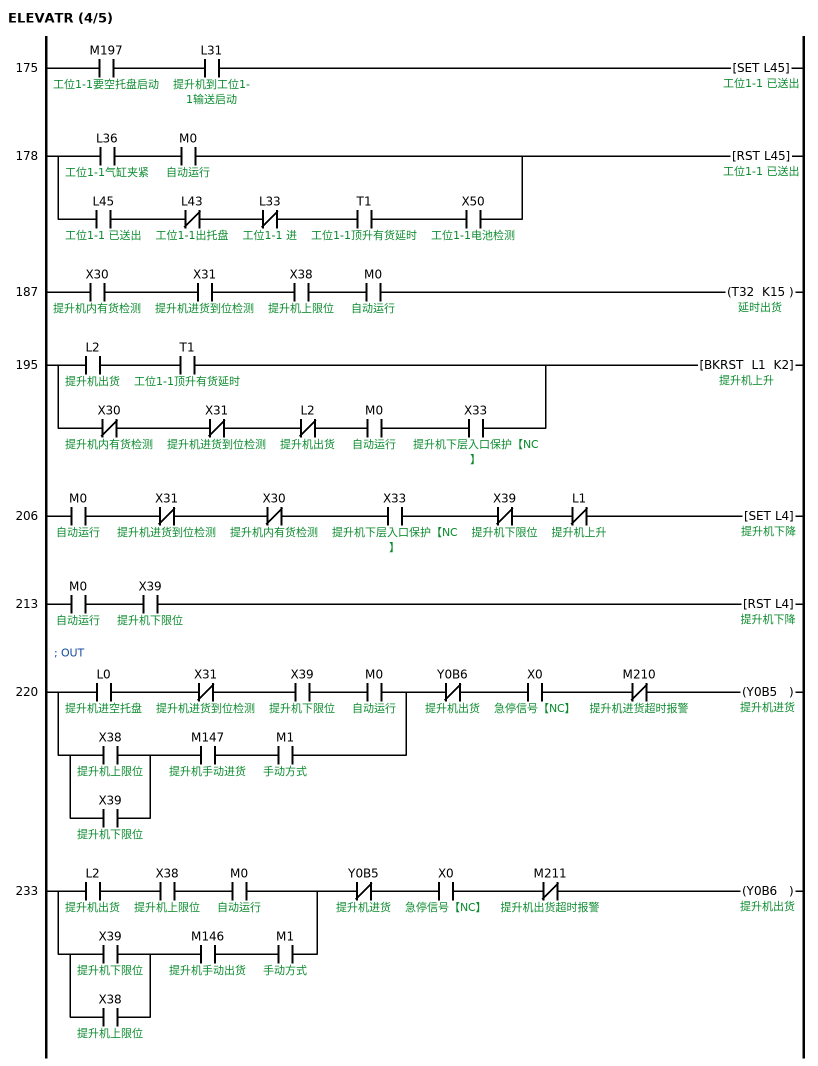
[picture p24: ladder of ELEVATR, rungs at steps 175 to 233]
175   LD      M197  ; 工位1-1要空托盘启动
      AND     L31  ; 提升机到工位1-1输送启动
      SET     L45  ; 工位1-1 已送出
178   LD      L36  ; 工位1-1气缸夹紧
      AND     M0  ; 自动运行
      LD      L45  ; 工位1-1 已送出
      ANI     L43  ; 工位1-1出托盘
      ANI     L33  ; 工位1-1 进
      AND     T1  ; 工位1-1顶升有货延时
      AND     X50  ; 工位1-1电池检测
      ORB
      RST     L45  ; 工位1-1 已送出
187   LD      X30  ; 提升机内有货检测
      AND     X31  ; 提升机进货到位检测
      AND     X38  ; 提升机上限位
      AND     M0  ; 自动运行
      OUT     T32 K15  ; 延时出货
195   LD      L2  ; 提升机出货
      AND     T1  ; 工位1-1顶升有货延时
      LDI     X30  ; 提升机内有货检测
      ANI     X31  ; 提升机进货到位检测
      ANI     L2  ; 提升机出货
      AND     M0  ; 自动运行
      AND     X33  ; 提升机下层入口保护【NC】
      ORB
      BKRST   L1 K2
206   LD      M0  ; 自动运行
      ANI     X31  ; 提升机进货到位检测
      ANI     X30  ; 提升机内有货检测
      AND     X33  ; 提升机下层入口保护【NC】
      ANI     X39  ; 提升机下限位
      ANI     L1  ; 提升机上升
      SET     L4  ; 提升机下降
213   LD      M0  ; 自动运行
      AND     X39  ; 提升机下限位
      RST     L4  ; 提升机下降
; OUT
220   LD      L0  ; 提升机进空托盘
      ANI     X31  ; 提升机进货到位检测
      AND     X39  ; 提升机下限位
      AND     M0  ; 自动运行
      LD      X38  ; 提升机上限位
      OR      X39  ; 提升机下限位
      AND     M147  ; 提升机手动进货
      AND     M1  ; 手动方式
      ORB
      ANI     Y0B6  ; 提升机出货
      AND     X0  ; 急停信号【NC】
      ANI     M210  ; 提升机进货超时报警
      OUT     Y0B5  ; 提升机进货
233   LD      L2  ; 提升机出货
      AND     X38  ; 提升机上限位
      AND     M0  ; 自动运行
      LD      X39  ; 提升机下限位
      OR      X38  ; 提升机上限位
      AND     M146  ; 提升机手动出货
      AND     M1  ; 手动方式
      ORB
      ANI     Y0B5  ; 提升机进货
      AND     X0  ; 急停信号【NC】
      ANI     M211  ; 提升机出货超时报警
      OUT     Y0B6  ; 提升机出货
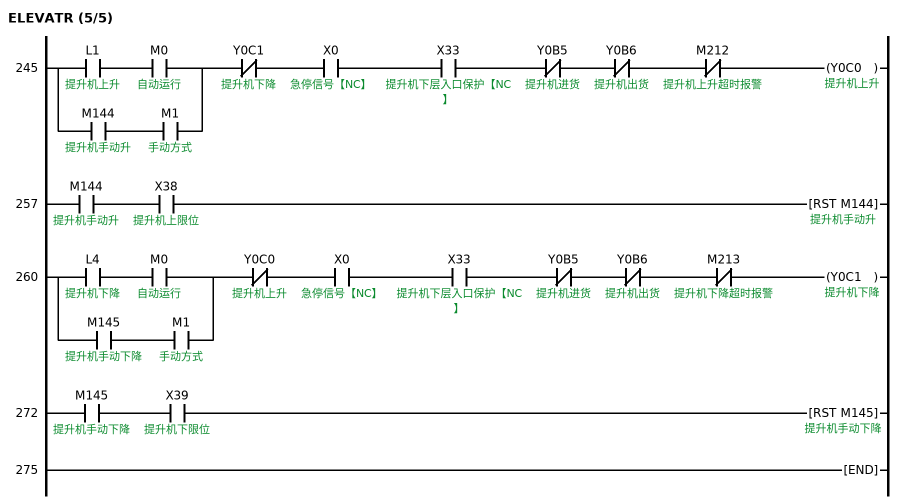
245   LD      L1  ; 提升机上升
      AND     M0  ; 自动运行
      LD      M144  ; 提升机手动升
      AND     M1  ; 手动方式
      ORB
      ANI     Y0C1  ; 提升机下降
      AND     X0  ; 急停信号【NC】
      AND     X33  ; 提升机下层入口保护【NC】
      ANI     Y0B5  ; 提升机进货
      ANI     Y0B6  ; 提升机出货
      ANI     M212  ; 提升机上升超时报警
      OUT     Y0C0  ; 提升机上升
257   LD      M144  ; 提升机手动升
      AND     X38  ; 提升机上限位
      RST     M144  ; 提升机手动升
260   LD      L4  ; 提升机下降
      AND     M0  ; 自动运行
      LD      M145  ; 提升机手动下降
      AND     M1  ; 手动方式
      ORB
      ANI     Y0C0  ; 提升机上升
      AND     X0  ; 急停信号【NC】
      AND     X33  ; 提升机下层入口保护【NC】
      ANI     Y0B5  ; 提升机进货
      ANI     Y0B6  ; 提升机出货
      ANI     M213  ; 提升机下降超时报警
      OUT     Y0C1  ; 提升机下降
272   LD      M145  ; 提升机手动下降
      AND     X39  ; 提升机下限位
      RST     M145  ; 提升机手动下降
275   END
END_PROGRAM

PROGRAM STATION1
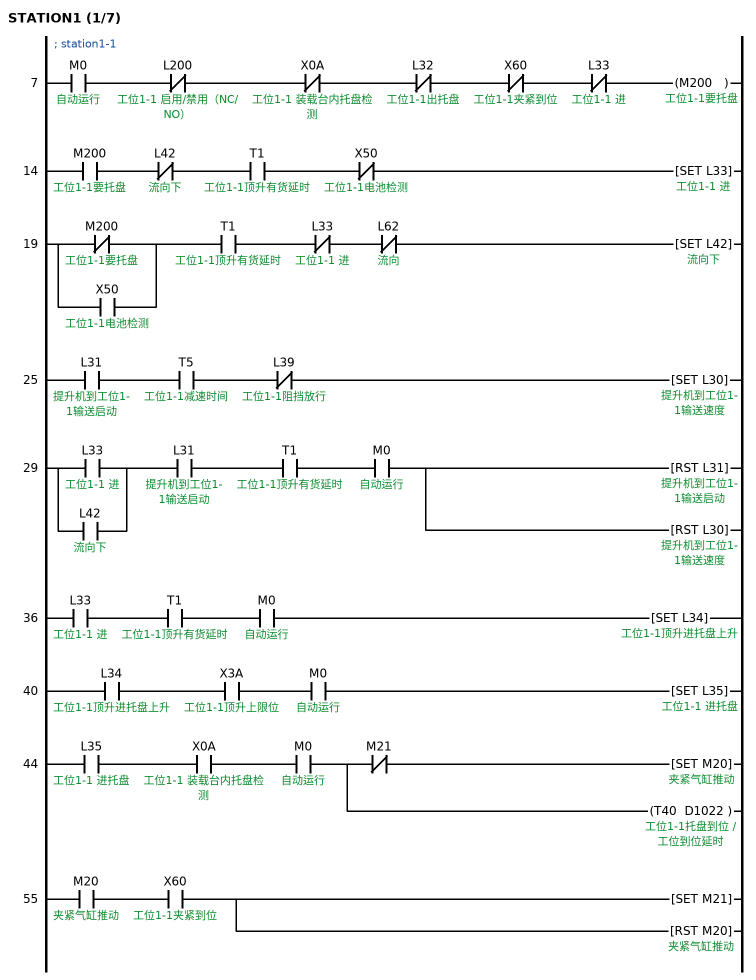
; station1-1
7     LD      M0  ; 自动运行
      ANI     L200  ; 工位1-1 启用/禁用（NC/NO）
      ANI     X0A  ; 工位1-1 装载台内托盘检测
      ANI     L32  ; 工位1-1出托盘
      ANI     X60  ; 工位1-1夹紧到位
      ANI     L33  ; 工位1-1 进
      OUT     M200  ; 工位1-1要托盘
14    LD      M200  ; 工位1-1要托盘
      ANI     L42  ; 流向下
      AND     T1  ; 工位1-1顶升有货延时
      ANI     X50  ; 工位1-1电池检测
      SET     L33  ; 工位1-1 进
19    LDI     M200  ; 工位1-1要托盘
      OR      X50  ; 工位1-1电池检测
      AND     T1  ; 工位1-1顶升有货延时
      ANI     L33  ; 工位1-1 进
      ANI     L62  ; 流向
      SET     L42  ; 流向下
25    LD      L31  ; 提升机到工位1-1输送启动
      AND     T5  ; 工位1-1减速时间
      ANI     L39  ; 工位1-1阻挡放行
      SET     L30  ; 提升机到工位1-1输送速度
29    LD      L33  ; 工位1-1 进
      OR      L42  ; 流向下
      AND     L31  ; 提升机到工位1-1输送启动
      AND     T1  ; 工位1-1顶升有货延时
      AND     M0  ; 自动运行
      RST     L31  ; 提升机到工位1-1输送启动
      RST     L30  ; 提升机到工位1-1输送速度
36    LD      L33  ; 工位1-1 进
      AND     T1  ; 工位1-1顶升有货延时
      AND     M0  ; 自动运行
      SET     L34  ; 工位1-1顶升进托盘上升
40    LD      L34  ; 工位1-1顶升进托盘上升
      AND     X3A  ; 工位1-1顶升上限位
      AND     M0  ; 自动运行
      SET     L35  ; 工位1-1 进托盘
44    LD      L35  ; 工位1-1 进托盘
      AND     X0A  ; 工位1-1 装载台内托盘检测
      AND     M0  ; 自动运行
      MPS
      ANI     M21
      SET     M20  ; 夹紧气缸推动
      MPP
      OUT     T40 D1022  ; 工位1-1托盘到位 / 工位到位延时
55    LD      M20  ; 夹紧气缸推动
      AND     X60  ; 工位1-1夹紧到位
      SET     M21
      RST     M20  ; 夹紧气缸推动
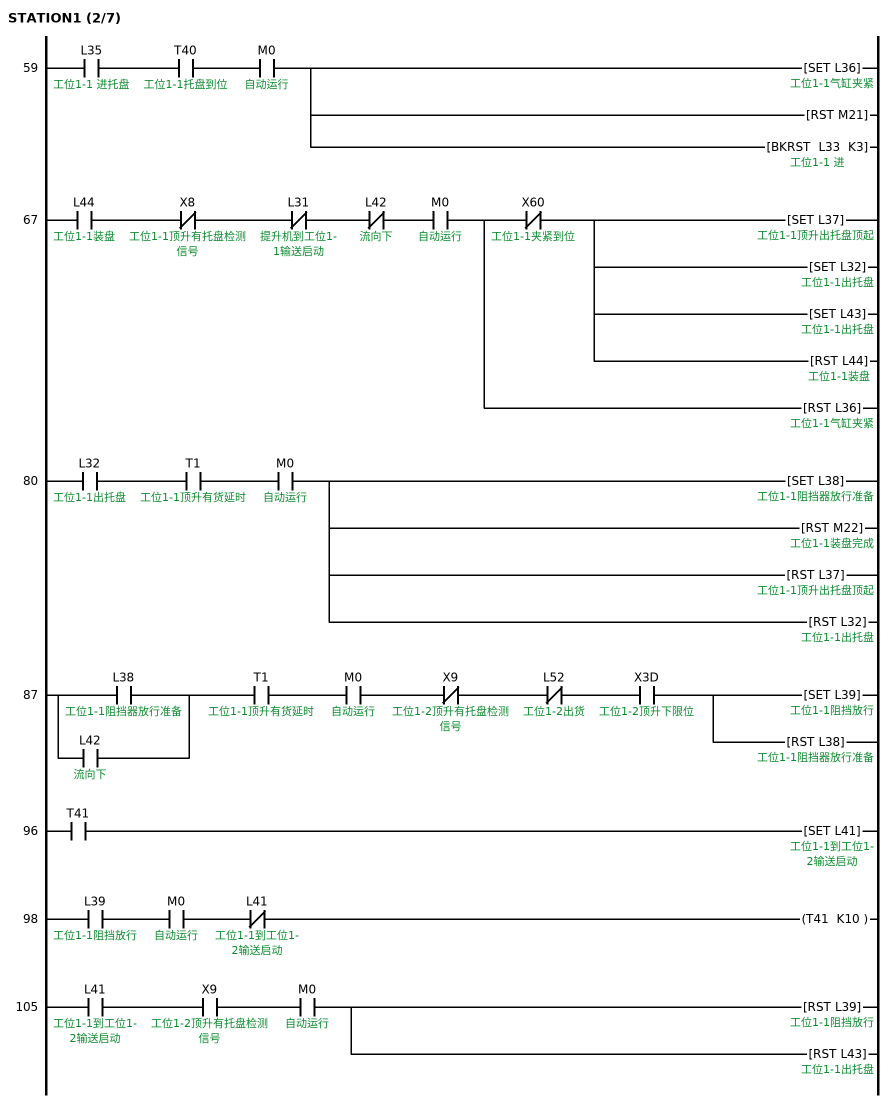
59    LD      L35  ; 工位1-1 进托盘
      AND     T40  ; 工位1-1托盘到位
      AND     M0  ; 自动运行
      SET     L36  ; 工位1-1气缸夹紧
      RST     M21
      BKRST   L33 K3
67    LD      L44  ; 工位1-1装盘
      ANI     X8  ; 工位1-1顶升有托盘检测信号
      ANI     L31  ; 提升机到工位1-1输送启动
      ANI     L42  ; 流向下
      AND     M0  ; 自动运行
      MPS
      ANI     X60  ; 工位1-1夹紧到位
      SET     L37  ; 工位1-1顶升出托盘顶起
      SET     L32  ; 工位1-1出托盘
      SET     L43  ; 工位1-1出托盘
      RST     L44  ; 工位1-1装盘
      MPP
      RST     L36  ; 工位1-1气缸夹紧
80    LD      L32  ; 工位1-1出托盘
      AND     T1  ; 工位1-1顶升有货延时
      AND     M0  ; 自动运行
      SET     L38  ; 工位1-1阻挡器放行准备
      RST     M22  ; 工位1-1装盘完成
      RST     L37  ; 工位1-1顶升出托盘顶起
      RST     L32  ; 工位1-1出托盘
87    LD      L38  ; 工位1-1阻挡器放行准备
      OR      L42  ; 流向下
      AND     T1  ; 工位1-1顶升有货延时
      AND     M0  ; 自动运行
      ANI     X9  ; 工位1-2顶升有托盘检测信号
      ANI     L52  ; 工位1-2出货
      AND     X3D  ; 工位1-2顶升下限位
      SET     L39  ; 工位1-1阻挡放行
      RST     L38  ; 工位1-1阻挡器放行准备
96    LD      T41
      SET     L41  ; 工位1-1到工位1-2输送启动
98    LD      L39  ; 工位1-1阻挡放行
      AND     M0  ; 自动运行
      ANI     L41  ; 工位1-1到工位1-2输送启动
      OUT     T41 K10
105   LD      L41  ; 工位1-1到工位1-2输送启动
      AND     X9  ; 工位1-2顶升有托盘检测信号
      AND     M0  ; 自动运行
      RST     L39  ; 工位1-1阻挡放行
      RST     L43  ; 工位1-1出托盘
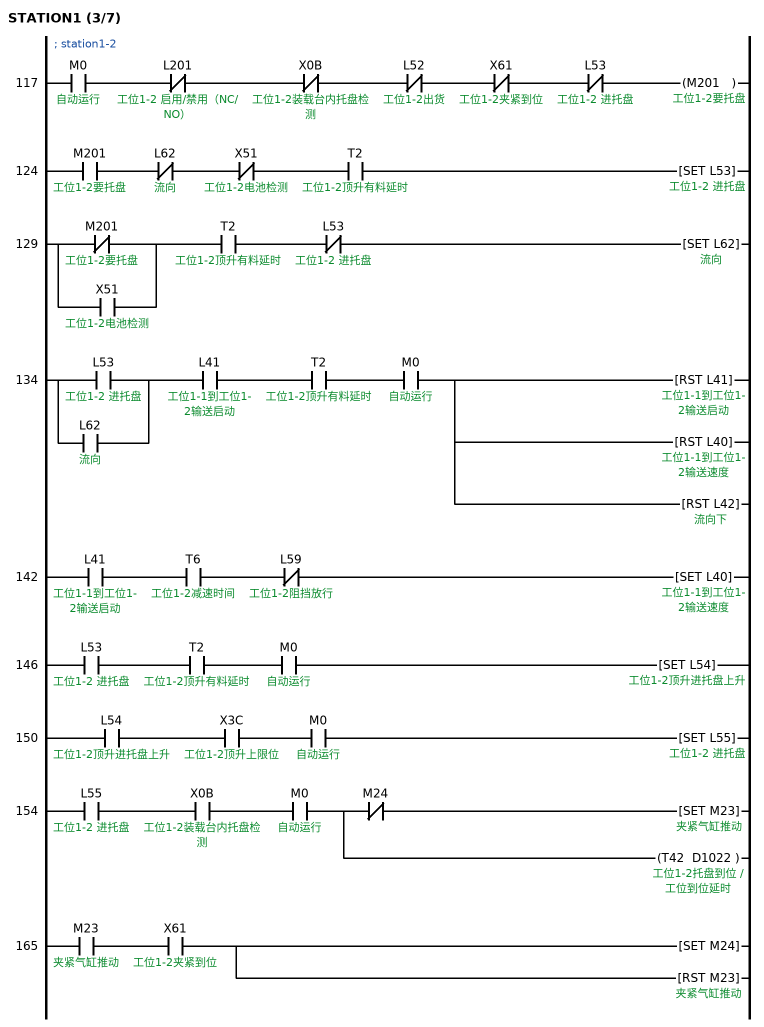
; station1-2
117   LD      M0  ; 自动运行
      ANI     L201  ; 工位1-2 启用/禁用（NC/NO）
      ANI     X0B  ; 工位1-2装载台内托盘检测
      ANI     L52  ; 工位1-2出货
      ANI     X61  ; 工位1-2夹紧到位
      ANI     L53  ; 工位1-2 进托盘
      OUT     M201  ; 工位1-2要托盘
124   LD      M201  ; 工位1-2要托盘
      ANI     L62  ; 流向
      ANI     X51  ; 工位1-2电池检测
      AND     T2  ; 工位1-2顶升有料延时
      SET     L53  ; 工位1-2 进托盘
129   LDI     M201  ; 工位1-2要托盘
      OR      X51  ; 工位1-2电池检测
      AND     T2  ; 工位1-2顶升有料延时
      ANI     L53  ; 工位1-2 进托盘
      SET     L62  ; 流向
134   LD      L53  ; 工位1-2 进托盘
      OR      L62  ; 流向
      AND     L41  ; 工位1-1到工位1-2输送启动
      AND     T2  ; 工位1-2顶升有料延时
      AND     M0  ; 自动运行
      RST     L41  ; 工位1-1到工位1-2输送启动
      RST     L40  ; 工位1-1到工位1-2输送速度
      RST     L42  ; 流向下
142   LD      L41  ; 工位1-1到工位1-2输送启动
      AND     T6  ; 工位1-2减速时间
      ANI     L59  ; 工位1-2阻挡放行
      SET     L40  ; 工位1-1到工位1-2输送速度
146   LD      L53  ; 工位1-2 进托盘
      AND     T2  ; 工位1-2顶升有料延时
      AND     M0  ; 自动运行
      SET     L54  ; 工位1-2顶升进托盘上升
150   LD      L54  ; 工位1-2顶升进托盘上升
      AND     X3C  ; 工位1-2顶升上限位
      AND     M0  ; 自动运行
      SET     L55  ; 工位1-2 进托盘
154   LD      L55  ; 工位1-2 进托盘
      AND     X0B  ; 工位1-2装载台内托盘检测
      AND     M0  ; 自动运行
      MPS
      ANI     M24
      SET     M23  ; 夹紧气缸推动
      MPP
      OUT     T42 D1022  ; 工位1-2托盘到位 / 工位到位延时
165   LD      M23  ; 夹紧气缸推动
      AND     X61  ; 工位1-2夹紧到位
      SET     M24
      RST     M23  ; 夹紧气缸推动
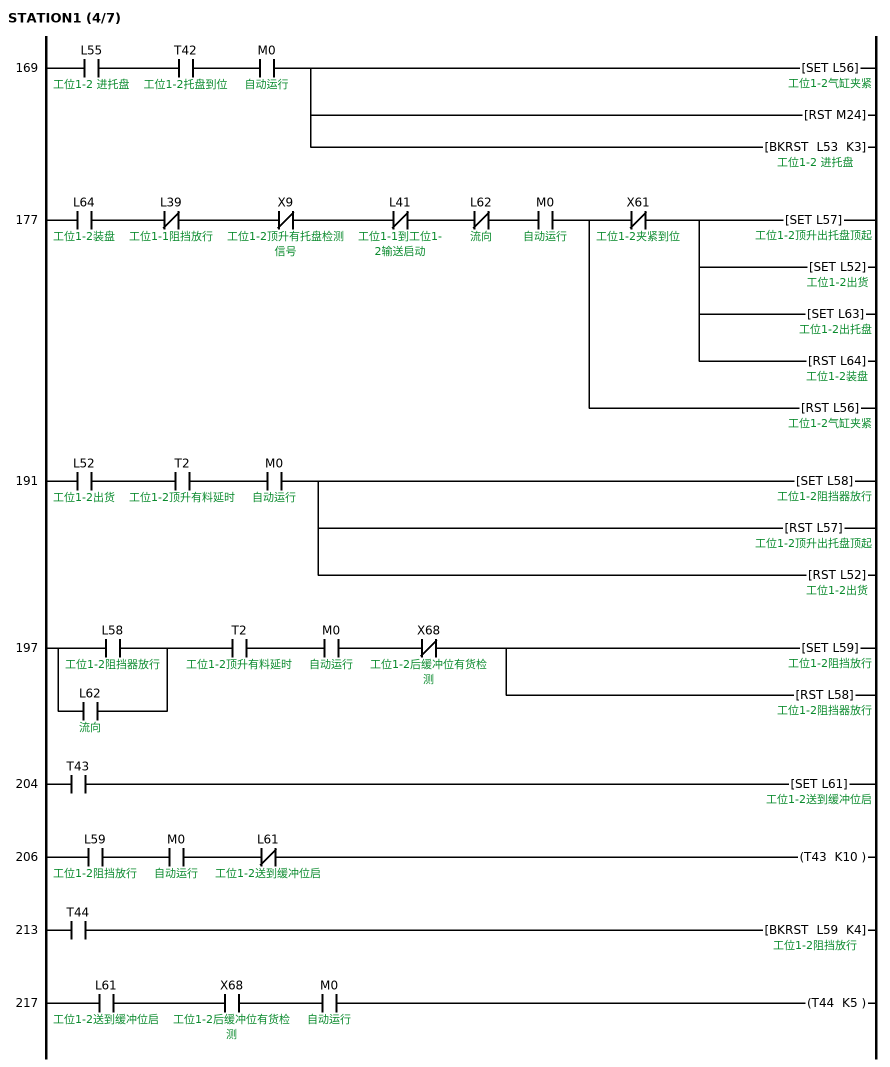
169   LD      L55  ; 工位1-2 进托盘
      AND     T42  ; 工位1-2托盘到位
      AND     M0  ; 自动运行
      SET     L56  ; 工位1-2气缸夹紧
      RST     M24
      BKRST   L53 K3
177   LD      L64  ; 工位1-2装盘
      ANI     L39  ; 工位1-1阻挡放行
      ANI     X9  ; 工位1-2顶升有托盘检测信号
      ANI     L41  ; 工位1-1到工位1-2输送启动
      ANI     L62  ; 流向
      AND     M0  ; 自动运行
      MPS
      ANI     X61  ; 工位1-2夹紧到位
      SET     L57  ; 工位1-2顶升出托盘顶起
      SET     L52  ; 工位1-2出货
      SET     L63  ; 工位1-2出托盘
      RST     L64  ; 工位1-2装盘
      MPP
      RST     L56  ; 工位1-2气缸夹紧
191   LD      L52  ; 工位1-2出货
      AND     T2  ; 工位1-2顶升有料延时
      AND     M0  ; 自动运行
      SET     L58  ; 工位1-2阻挡器放行
      RST     L57  ; 工位1-2顶升出托盘顶起
      RST     L52  ; 工位1-2出货
197   LD      L58  ; 工位1-2阻挡器放行
      OR      L62  ; 流向
      AND     T2  ; 工位1-2顶升有料延时
      AND     M0  ; 自动运行
      ANI     X68  ; 工位1-2后缓冲位有货检测
      SET     L59  ; 工位1-2阻挡放行
      RST     L58  ; 工位1-2阻挡器放行
204   LD      T43
      SET     L61  ; 工位1-2送到缓冲位启
206   LD      L59  ; 工位1-2阻挡放行
      AND     M0  ; 自动运行
      ANI     L61  ; 工位1-2送到缓冲位启
      OUT     T43 K10
213   LD      T44
      BKRST   L59 K4
217   LD      L61  ; 工位1-2送到缓冲位启
      AND     X68  ; 工位1-2后缓冲位有货检测
      AND     M0  ; 自动运行
      OUT     T44 K5
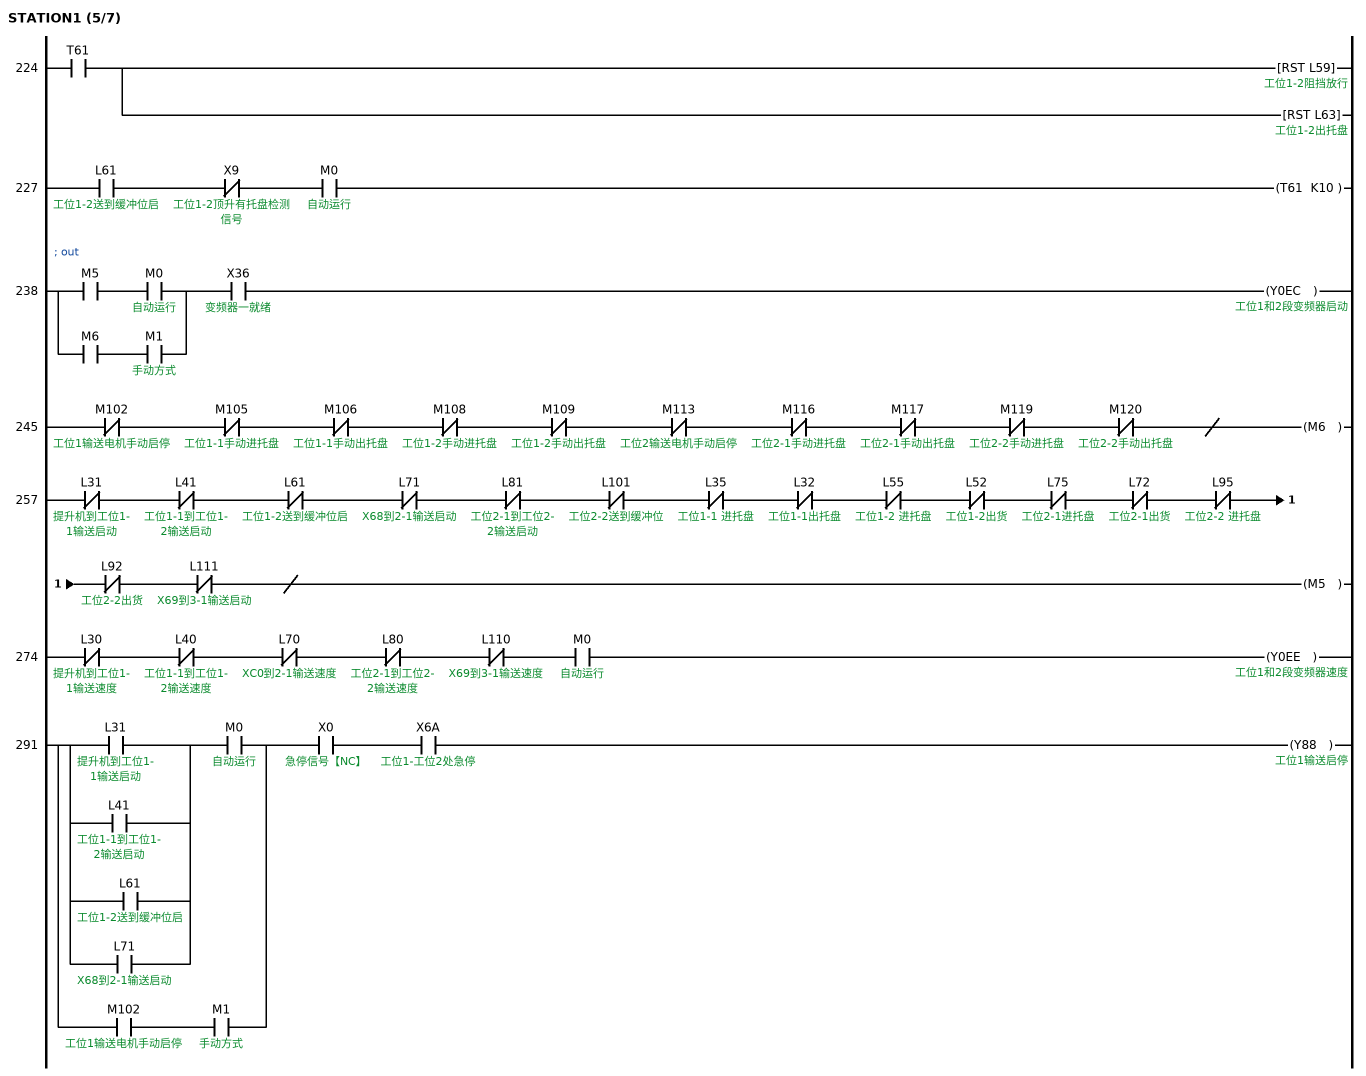
224   LD      T61
      RST     L59  ; 工位1-2阻挡放行
      RST     L63  ; 工位1-2出托盘
227   LD      L61  ; 工位1-2送到缓冲位启
      ANI     X9  ; 工位1-2顶升有托盘检测信号
      AND     M0  ; 自动运行
      OUT     T61 K10
; out
238   LD      M5
      AND     M0  ; 自动运行
      LD      M6
      AND     M1  ; 手动方式
      ORB
      AND     X36  ; 变频器一就绪
      OUT     Y0EC  ; 工位1和2段变频器启动
245   LDI     M102  ; 工位1输送电机手动启停
      ANI     M105  ; 工位1-1手动进托盘
      ANI     M106  ; 工位1-1手动出托盘
      ANI     M108  ; 工位1-2手动进托盘
      ANI     M109  ; 工位1-2手动出托盘
      ANI     M113  ; 工位2输送电机手动启停
      ANI     M116  ; 工位2-1手动进托盘
      ANI     M117  ; 工位2-1手动出托盘
      ANI     M119  ; 工位2-2手动进托盘
      ANI     M120  ; 工位2-2手动出托盘
      INV
      OUT     M6
257   LDI     L31  ; 提升机到工位1-1输送启动
      ANI     L41  ; 工位1-1到工位1-2输送启动
      ANI     L61  ; 工位1-2送到缓冲位启
      ANI     L71  ; X68到2-1输送启动
      ANI     L81  ; 工位2-1到工位2-2输送启动
      ANI     L101  ; 工位2-2送到缓冲位
      ANI     L35  ; 工位1-1 进托盘
      ANI     L32  ; 工位1-1出托盘
      ANI     L55  ; 工位1-2 进托盘
      ANI     L52  ; 工位1-2出货
      ANI     L75  ; 工位2-1进托盘
      ANI     L72  ; 工位2-1出货
      ANI     L95  ; 工位2-2 进托盘
      ANI     L92  ; 工位2-2出货
      ANI     L111  ; X69到3-1输送启动
      INV
      OUT     M5
274   LDI     L30  ; 提升机到工位1-1输送速度
      ANI     L40  ; 工位1-1到工位1-2输送速度
      ANI     L70  ; XC0到2-1输送速度
      ANI     L80  ; 工位2-1到工位2-2输送速度
      ANI     L110  ; X69到3-1输送速度
      AND     M0  ; 自动运行
      OUT     Y0EE  ; 工位1和2段变频器速度
        [note] ON高速，OFF低速
291   LD      L31  ; 提升机到工位1-1输送启动
      OR      L41  ; 工位1-1到工位1-2输送启动
      OR      L61  ; 工位1-2送到缓冲位启
      OR      L71  ; X68到2-1输送启动
      AND     M0  ; 自动运行
      LD      M102  ; 工位1输送电机手动启停
      AND     M1  ; 手动方式
      ORB
      AND     X0  ; 急停信号【NC】
      AND     X6A  ; 工位1-工位2处急停
      OUT     Y88  ; 工位1输送启停
        [note] 1-1
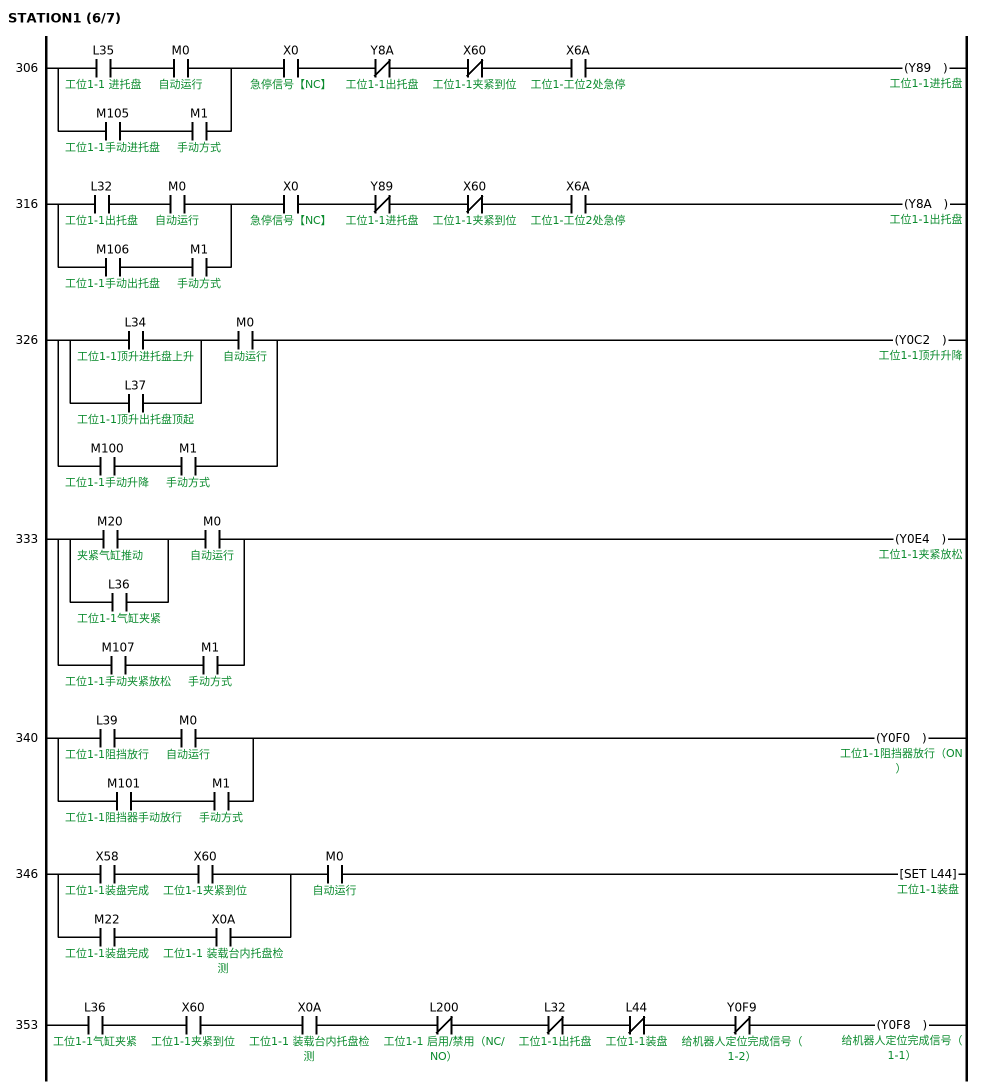
306   LD      L35  ; 工位1-1 进托盘
      AND     M0  ; 自动运行
      LD      M105  ; 工位1-1手动进托盘
      AND     M1  ; 手动方式
      ORB
      AND     X0  ; 急停信号【NC】
      ANI     Y8A  ; 工位1-1出托盘
      ANI     X60  ; 工位1-1夹紧到位
      AND     X6A  ; 工位1-工位2处急停
      OUT     Y89  ; 工位1-1进托盘
316   LD      L32  ; 工位1-1出托盘
      AND     M0  ; 自动运行
      LD      M106  ; 工位1-1手动出托盘
      AND     M1  ; 手动方式
      ORB
      AND     X0  ; 急停信号【NC】
      ANI     Y89  ; 工位1-1进托盘
      ANI     X60  ; 工位1-1夹紧到位
      AND     X6A  ; 工位1-工位2处急停
      OUT     Y8A  ; 工位1-1出托盘
326   LD      L34  ; 工位1-1顶升进托盘上升
      OR      L37  ; 工位1-1顶升出托盘顶起
      AND     M0  ; 自动运行
      LD      M100  ; 工位1-1手动升降
      AND     M1  ; 手动方式
      ORB
      OUT     Y0C2  ; 工位1-1顶升升降
333   LD      M20  ; 夹紧气缸推动
      OR      L36  ; 工位1-1气缸夹紧
      AND     M0  ; 自动运行
      LD      M107  ; 工位1-1手动夹紧放松
      AND     M1  ; 手动方式
      ORB
      OUT     Y0E4  ; 工位1-1夹紧放松
340   LD      L39  ; 工位1-1阻挡放行
      AND     M0  ; 自动运行
      LD      M101  ; 工位1-1阻挡器手动放行
      AND     M1  ; 手动方式
      ORB
      OUT     Y0F0  ; 工位1-1阻挡器放行（ON）
346   LD      X58  ; 工位1-1装盘完成
      AND     X60  ; 工位1-1夹紧到位
      LD      M22  ; 工位1-1装盘完成
      AND     X0A  ; 工位1-1 装载台内托盘检测
      ORB
      AND     M0  ; 自动运行
      SET     L44  ; 工位1-1装盘
353   LD      L36  ; 工位1-1气缸夹紧
      AND     X60  ; 工位1-1夹紧到位
      AND     X0A  ; 工位1-1 装载台内托盘检测
      ANI     L200  ; 工位1-1 启用/禁用（NC/NO）
      ANI     L32  ; 工位1-1出托盘
      ANI     L44  ; 工位1-1装盘
      ANI     Y0F9  ; 给机器人定位完成信号（1-2）
      OUT     Y0F8  ; 给机器人定位完成信号（1-1）
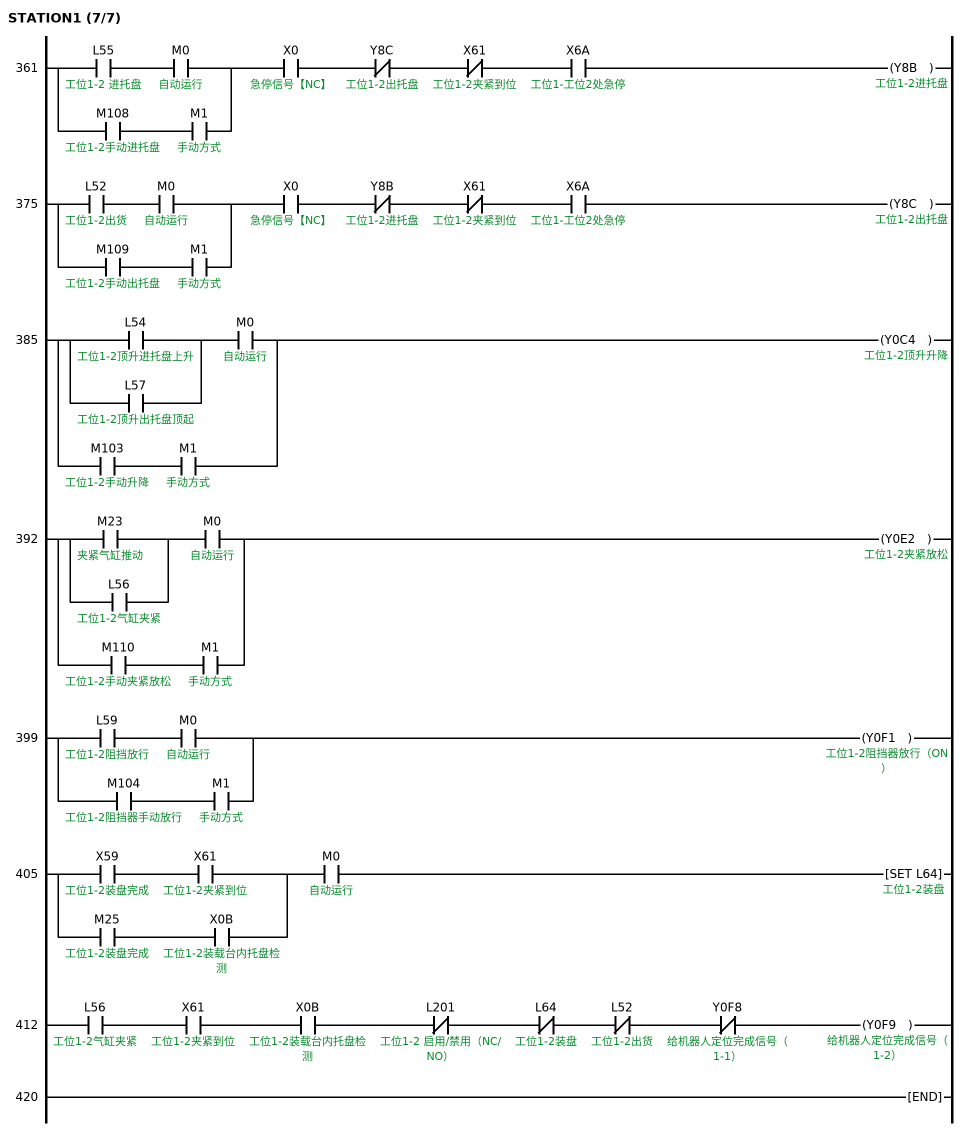
361   LD      L55  ; 工位1-2 进托盘
      AND     M0  ; 自动运行
      LD      M108  ; 工位1-2手动进托盘
      AND     M1  ; 手动方式
      ORB
      AND     X0  ; 急停信号【NC】
      ANI     Y8C  ; 工位1-2出托盘
      ANI     X61  ; 工位1-2夹紧到位
      AND     X6A  ; 工位1-工位2处急停
      OUT     Y8B  ; 工位1-2进托盘
        [note] 1-2
375   LD      L52  ; 工位1-2出货
      AND     M0  ; 自动运行
      LD      M109  ; 工位1-2手动出托盘
      AND     M1  ; 手动方式
      ORB
      AND     X0  ; 急停信号【NC】
      ANI     Y8B  ; 工位1-2进托盘
      ANI     X61  ; 工位1-2夹紧到位
      AND     X6A  ; 工位1-工位2处急停
      OUT     Y8C  ; 工位1-2出托盘
385   LD      L54  ; 工位1-2顶升进托盘上升
      OR      L57  ; 工位1-2顶升出托盘顶起
      AND     M0  ; 自动运行
      LD      M103  ; 工位1-2手动升降
      AND     M1  ; 手动方式
      ORB
      OUT     Y0C4  ; 工位1-2顶升升降
392   LD      M23  ; 夹紧气缸推动
      OR      L56  ; 工位1-2气缸夹紧
      AND     M0  ; 自动运行
      LD      M110  ; 工位1-2手动夹紧放松
      AND     M1  ; 手动方式
      ORB
      OUT     Y0E2  ; 工位1-2夹紧放松
399   LD      L59  ; 工位1-2阻挡放行
      AND     M0  ; 自动运行
      LD      M104  ; 工位1-2阻挡器手动放行
      AND     M1  ; 手动方式
      ORB
      OUT     Y0F1  ; 工位1-2阻挡器放行（ON）
405   LD      X59  ; 工位1-2装盘完成
      AND     X61  ; 工位1-2夹紧到位
      LD      M25  ; 工位1-2装盘完成
      AND     X0B  ; 工位1-2装载台内托盘检测
      ORB
      AND     M0  ; 自动运行
      SET     L64  ; 工位1-2装盘
412   LD      L56  ; 工位1-2气缸夹紧
      AND     X61  ; 工位1-2夹紧到位
      AND     X0B  ; 工位1-2装载台内托盘检测
      ANI     L201  ; 工位1-2 启用/禁用（NC/NO）
      ANI     L64  ; 工位1-2装盘
      ANI     L52  ; 工位1-2出货
      ANI     Y0F8  ; 给机器人定位完成信号（1-1）
      OUT     Y0F9  ; 给机器人定位完成信号（1-2）
420   END
END_PROGRAM

PROGRAM STATION2
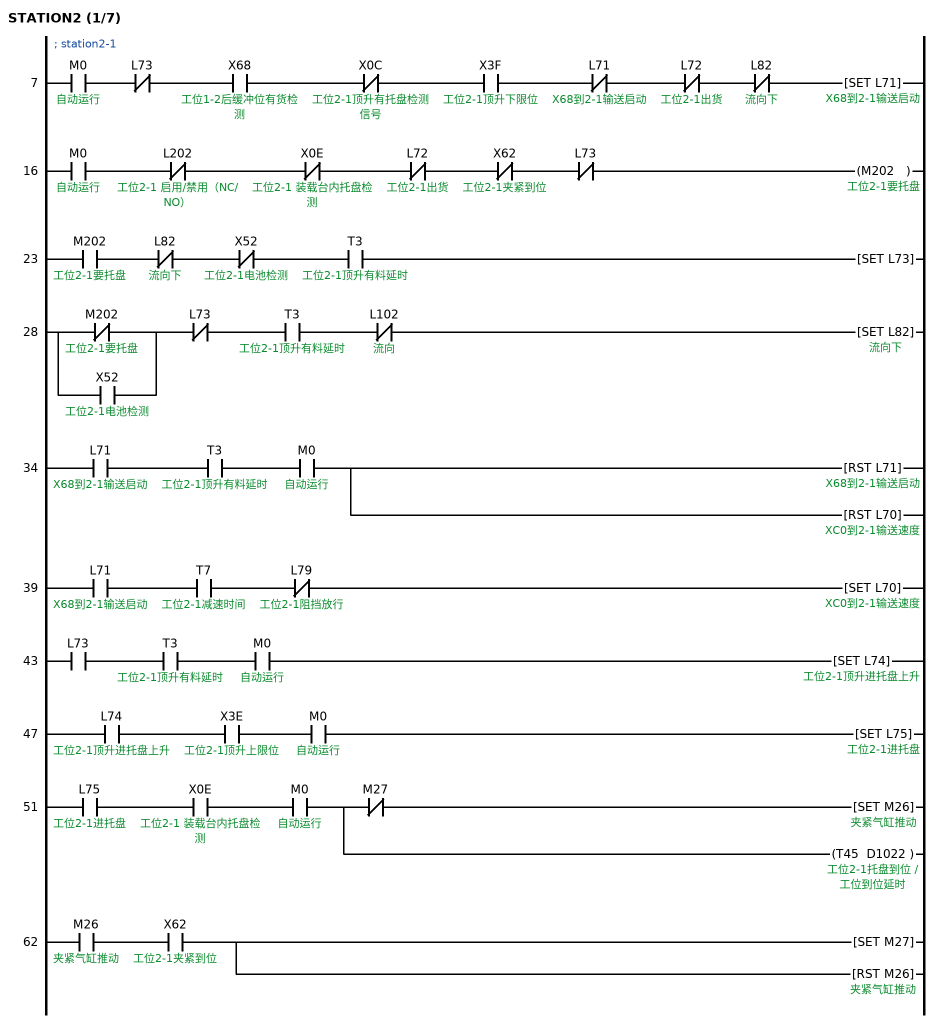
; station2-1
7     LD      M0  ; 自动运行
      ANI     L73
      AND     X68  ; 工位1-2后缓冲位有货检测
      ANI     X0C  ; 工位2-1顶升有托盘检测信号
      AND     X3F  ; 工位2-1顶升下限位
      ANI     L71  ; X68到2-1输送启动
      ANI     L72  ; 工位2-1出货
      ANI     L82  ; 流向下
      SET     L71  ; X68到2-1输送启动
16    LD      M0  ; 自动运行
      ANI     L202  ; 工位2-1 启用/禁用（NC/NO）
      ANI     X0E  ; 工位2-1 装载台内托盘检测
      ANI     L72  ; 工位2-1出货
      ANI     X62  ; 工位2-1夹紧到位
      ANI     L73
      OUT     M202  ; 工位2-1要托盘
23    LD      M202  ; 工位2-1要托盘
      ANI     L82  ; 流向下
      ANI     X52  ; 工位2-1电池检测
      AND     T3  ; 工位2-1顶升有料延时
      SET     L73
28    LDI     M202  ; 工位2-1要托盘
      OR      X52  ; 工位2-1电池检测
      ANI     L73
      AND     T3  ; 工位2-1顶升有料延时
      ANI     L102  ; 流向
      SET     L82  ; 流向下
34    LD      L71  ; X68到2-1输送启动
      AND     T3  ; 工位2-1顶升有料延时
      AND     M0  ; 自动运行
      RST     L71  ; X68到2-1输送启动
      RST     L70  ; XC0到2-1输送速度
39    LD      L71  ; X68到2-1输送启动
      AND     T7  ; 工位2-1减速时间
      ANI     L79  ; 工位2-1阻挡放行
      SET     L70  ; XC0到2-1输送速度
43    LD      L73
      AND     T3  ; 工位2-1顶升有料延时
      AND     M0  ; 自动运行
      SET     L74  ; 工位2-1顶升进托盘上升
47    LD      L74  ; 工位2-1顶升进托盘上升
      AND     X3E  ; 工位2-1顶升上限位
      AND     M0  ; 自动运行
      SET     L75  ; 工位2-1进托盘
51    LD      L75  ; 工位2-1进托盘
      AND     X0E  ; 工位2-1 装载台内托盘检测
      AND     M0  ; 自动运行
      MPS
      ANI     M27
      SET     M26  ; 夹紧气缸推动
      MPP
      OUT     T45 D1022  ; 工位2-1托盘到位 / 工位到位延时
62    LD      M26  ; 夹紧气缸推动
      AND     X62  ; 工位2-1夹紧到位
      SET     M27
      RST     M26  ; 夹紧气缸推动
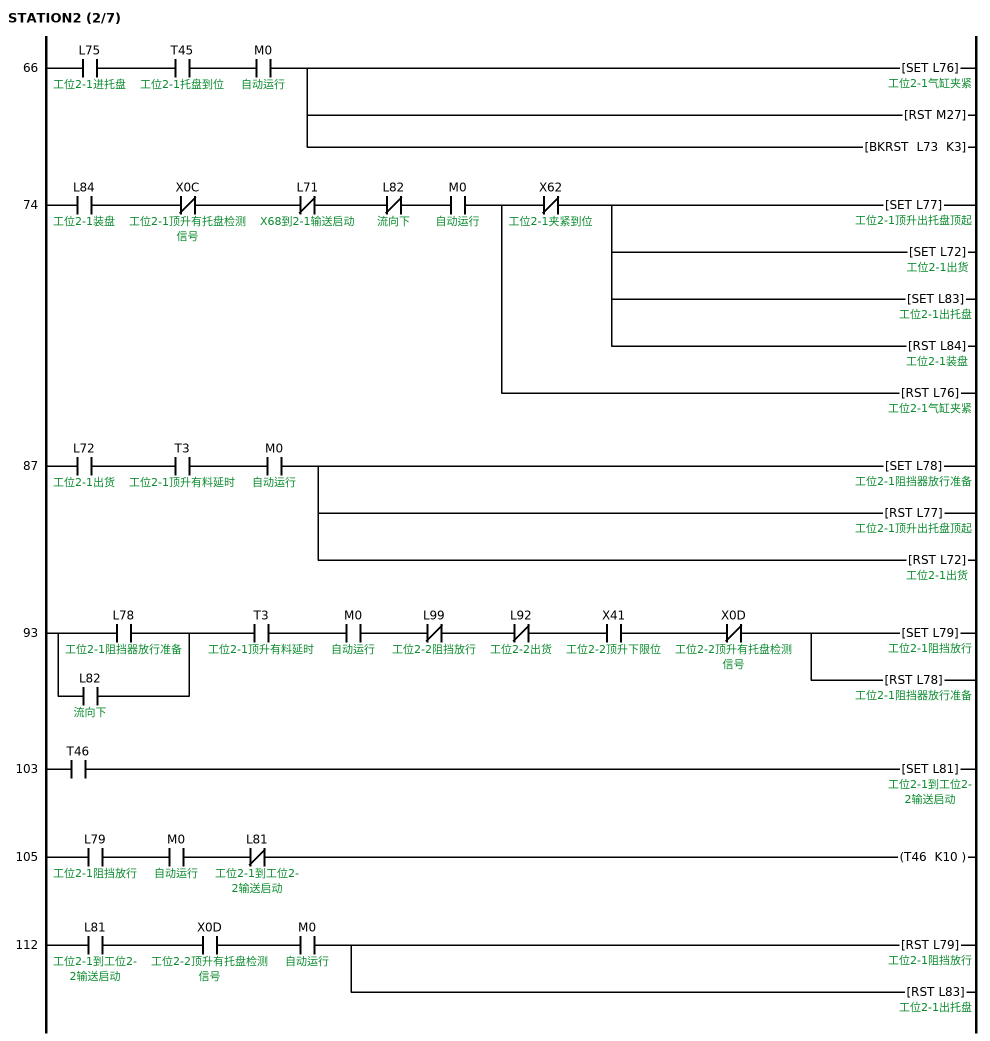
66    LD      L75  ; 工位2-1进托盘
      AND     T45  ; 工位2-1托盘到位
      AND     M0  ; 自动运行
      SET     L76  ; 工位2-1气缸夹紧
      RST     M27
      BKRST   L73 K3
74    LD      L84  ; 工位2-1装盘
      ANI     X0C  ; 工位2-1顶升有托盘检测信号
      ANI     L71  ; X68到2-1输送启动
      ANI     L82  ; 流向下
      AND     M0  ; 自动运行
      MPS
      ANI     X62  ; 工位2-1夹紧到位
      SET     L77  ; 工位2-1顶升出托盘顶起
      SET     L72  ; 工位2-1出货
      SET     L83  ; 工位2-1出托盘
      RST     L84  ; 工位2-1装盘
      MPP
      RST     L76  ; 工位2-1气缸夹紧
87    LD      L72  ; 工位2-1出货
      AND     T3  ; 工位2-1顶升有料延时
      AND     M0  ; 自动运行
      SET     L78  ; 工位2-1阻挡器放行准备
      RST     L77  ; 工位2-1顶升出托盘顶起
      RST     L72  ; 工位2-1出货
93    LD      L78  ; 工位2-1阻挡器放行准备
      OR      L82  ; 流向下
      AND     T3  ; 工位2-1顶升有料延时
      AND     M0  ; 自动运行
      ANI     L99  ; 工位2-2阻挡放行
      ANI     L92  ; 工位2-2出货
      AND     X41  ; 工位2-2顶升下限位
      ANI     X0D  ; 工位2-2顶升有托盘检测信号
      SET     L79  ; 工位2-1阻挡放行
      RST     L78  ; 工位2-1阻挡器放行准备
103   LD      T46
      SET     L81  ; 工位2-1到工位2-2输送启动
105   LD      L79  ; 工位2-1阻挡放行
      AND     M0  ; 自动运行
      ANI     L81  ; 工位2-1到工位2-2输送启动
      OUT     T46 K10
112   LD      L81  ; 工位2-1到工位2-2输送启动
      AND     X0D  ; 工位2-2顶升有托盘检测信号
      AND     M0  ; 自动运行
      RST     L79  ; 工位2-1阻挡放行
      RST     L83  ; 工位2-1出托盘
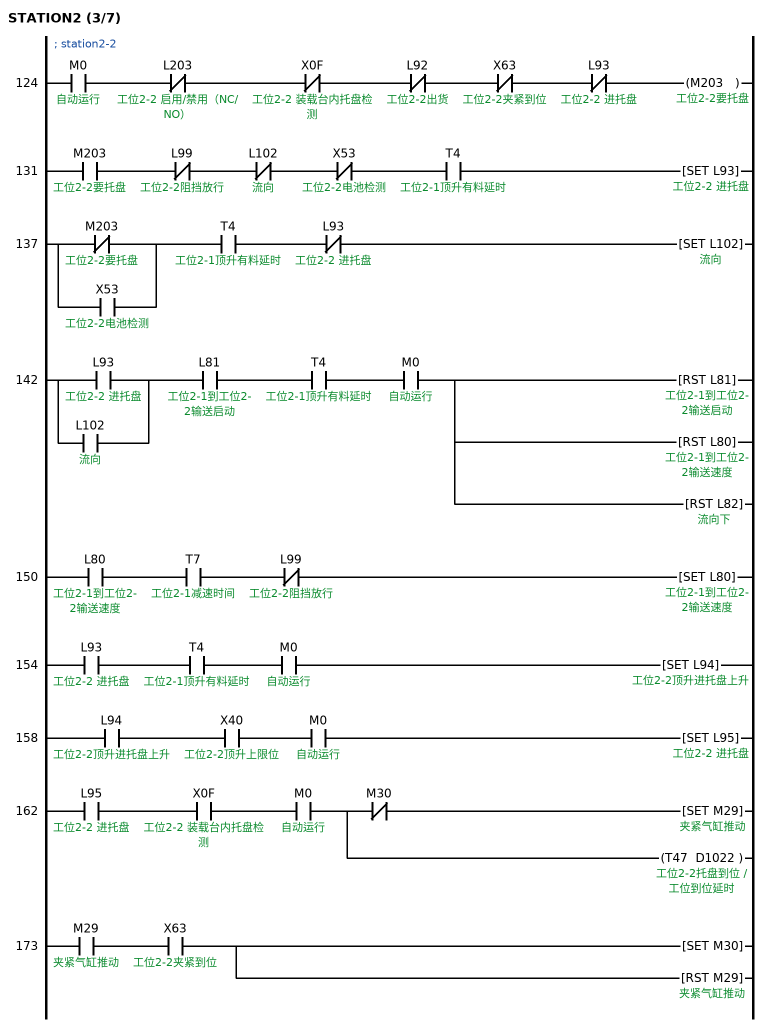
; station2-2
124   LD      M0  ; 自动运行
      ANI     L203  ; 工位2-2 启用/禁用（NC/NO）
      ANI     X0F  ; 工位2-2 装载台内托盘检测
      ANI     L92  ; 工位2-2出货
      ANI     X63  ; 工位2-2夹紧到位
      ANI     L93  ; 工位2-2 进托盘
      OUT     M203  ; 工位2-2要托盘
131   LD      M203  ; 工位2-2要托盘
      ANI     L99  ; 工位2-2阻挡放行
      ANI     L102  ; 流向
      ANI     X53  ; 工位2-2电池检测
      AND     T4  ; 工位2-1顶升有料延时
      SET     L93  ; 工位2-2 进托盘
137   LDI     M203  ; 工位2-2要托盘
      OR      X53  ; 工位2-2电池检测
      AND     T4  ; 工位2-1顶升有料延时
      ANI     L93  ; 工位2-2 进托盘
      SET     L102  ; 流向
142   LD      L93  ; 工位2-2 进托盘
      OR      L102  ; 流向
      AND     L81  ; 工位2-1到工位2-2输送启动
      AND     T4  ; 工位2-1顶升有料延时
      AND     M0  ; 自动运行
      RST     L81  ; 工位2-1到工位2-2输送启动
      RST     L80  ; 工位2-1到工位2-2输送速度
      RST     L82  ; 流向下
150   LD      L80  ; 工位2-1到工位2-2输送速度
      AND     T7  ; 工位2-1减速时间
      ANI     L99  ; 工位2-2阻挡放行
      SET     L80  ; 工位2-1到工位2-2输送速度
154   LD      L93  ; 工位2-2 进托盘
      AND     T4  ; 工位2-1顶升有料延时
      AND     M0  ; 自动运行
      SET     L94  ; 工位2-2顶升进托盘上升
158   LD      L94  ; 工位2-2顶升进托盘上升
      AND     X40  ; 工位2-2顶升上限位
      AND     M0  ; 自动运行
      SET     L95  ; 工位2-2 进托盘
162   LD      L95  ; 工位2-2 进托盘
      AND     X0F  ; 工位2-2 装载台内托盘检测
      AND     M0  ; 自动运行
      MPS
      ANI     M30
      SET     M29  ; 夹紧气缸推动
      MPP
      OUT     T47 D1022  ; 工位2-2托盘到位 / 工位到位延时
173   LD      M29  ; 夹紧气缸推动
      AND     X63  ; 工位2-2夹紧到位
      SET     M30
      RST     M29  ; 夹紧气缸推动
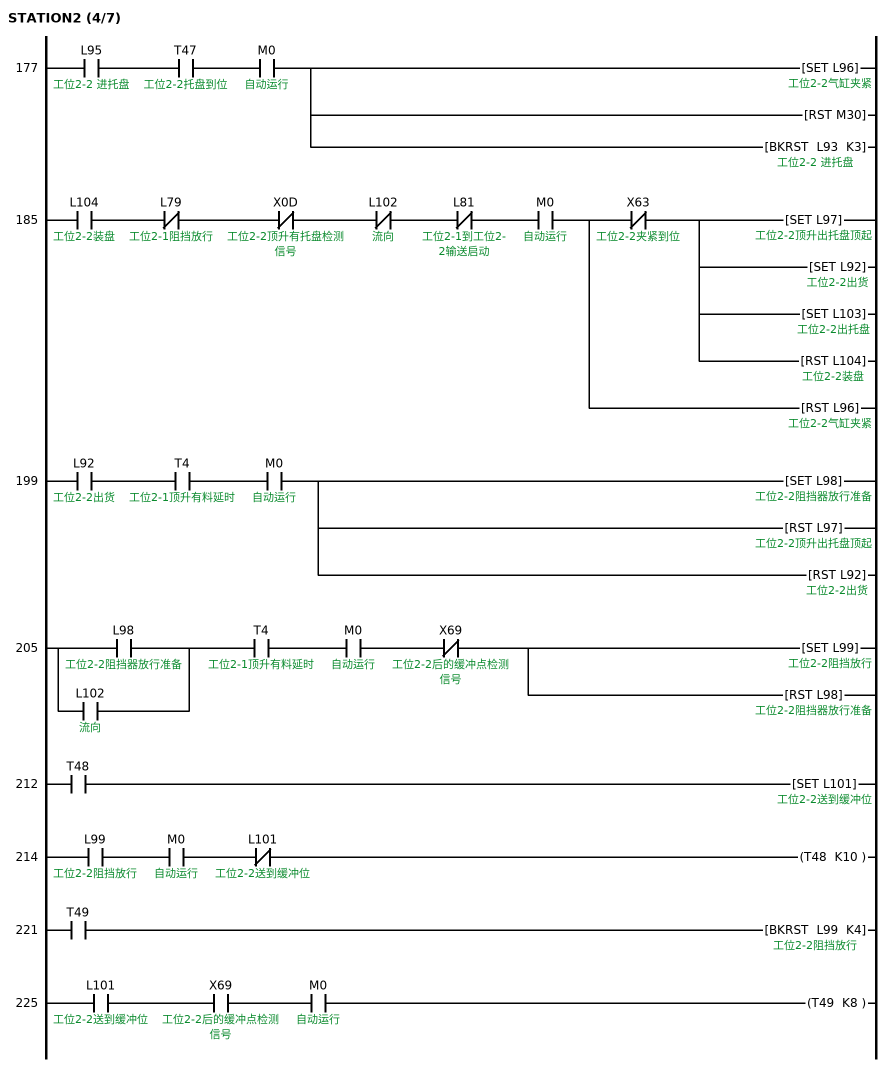
177   LD      L95  ; 工位2-2 进托盘
      AND     T47  ; 工位2-2托盘到位
      AND     M0  ; 自动运行
      SET     L96  ; 工位2-2气缸夹紧
      RST     M30
      BKRST   L93 K3
185   LD      L104  ; 工位2-2装盘
      ANI     L79  ; 工位2-1阻挡放行
      ANI     X0D  ; 工位2-2顶升有托盘检测信号
      ANI     L102  ; 流向
      ANI     L81  ; 工位2-1到工位2-2输送启动
      AND     M0  ; 自动运行
      MPS
      ANI     X63  ; 工位2-2夹紧到位
      SET     L97  ; 工位2-2顶升出托盘顶起
      SET     L92  ; 工位2-2出货
      SET     L103  ; 工位2-2出托盘
      RST     L104  ; 工位2-2装盘
      MPP
      RST     L96  ; 工位2-2气缸夹紧
199   LD      L92  ; 工位2-2出货
      AND     T4  ; 工位2-1顶升有料延时
      AND     M0  ; 自动运行
      SET     L98  ; 工位2-2阻挡器放行准备
      RST     L97  ; 工位2-2顶升出托盘顶起
      RST     L92  ; 工位2-2出货
205   LD      L98  ; 工位2-2阻挡器放行准备
      OR      L102  ; 流向
      AND     T4  ; 工位2-1顶升有料延时
      AND     M0  ; 自动运行
      ANI     X69  ; 工位2-2后的缓冲点检测信号
      SET     L99  ; 工位2-2阻挡放行
      RST     L98  ; 工位2-2阻挡器放行准备
212   LD      T48
      SET     L101  ; 工位2-2送到缓冲位
214   LD      L99  ; 工位2-2阻挡放行
      AND     M0  ; 自动运行
      ANI     L101  ; 工位2-2送到缓冲位
      OUT     T48 K10
221   LD      T49
      BKRST   L99 K4
225   LD      L101  ; 工位2-2送到缓冲位
      AND     X69  ; 工位2-2后的缓冲点检测信号
      AND     M0  ; 自动运行
      OUT     T49 K8
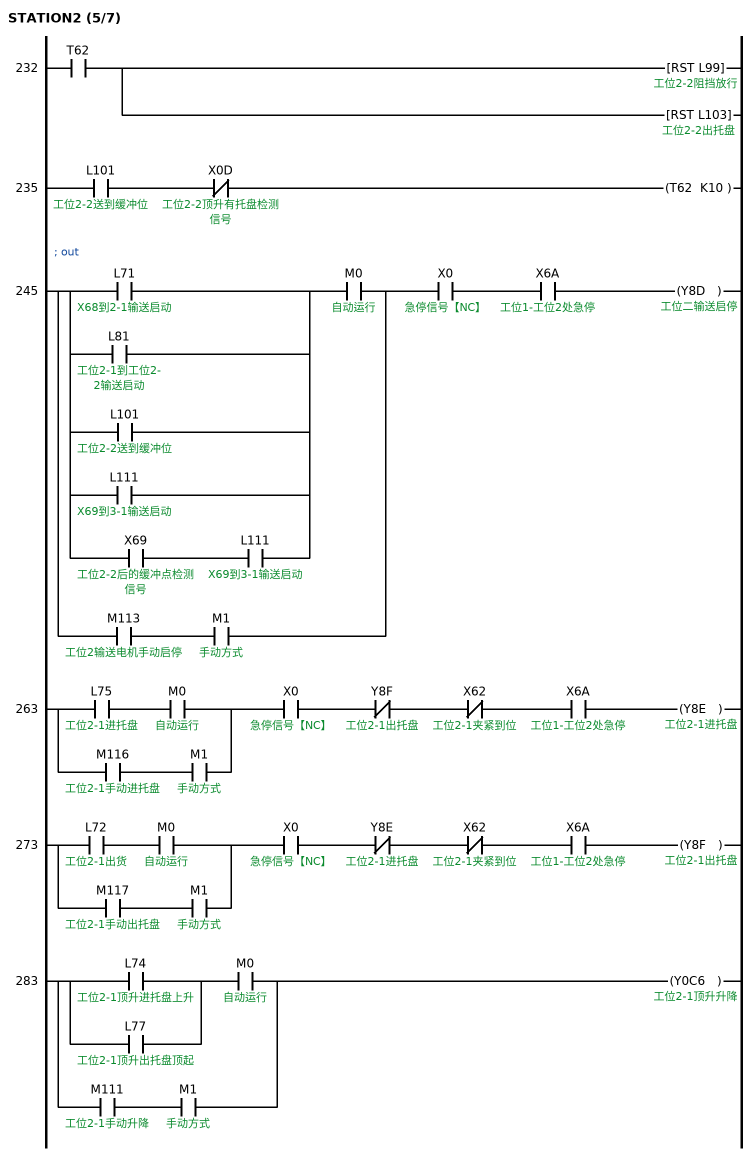
232   LD      T62
      RST     L99  ; 工位2-2阻挡放行
      RST     L103  ; 工位2-2出托盘
235   LD      L101  ; 工位2-2送到缓冲位
      ANI     X0D  ; 工位2-2顶升有托盘检测信号
      OUT     T62 K10
; out
245   LD      L71  ; X68到2-1输送启动
      OR      L81  ; 工位2-1到工位2-2输送启动
      OR      L101  ; 工位2-2送到缓冲位
      OR      L111  ; X69到3-1输送启动
      LD      X69  ; 工位2-2后的缓冲点检测信号
      AND     L111  ; X69到3-1输送启动
      ORB
      AND     M0  ; 自动运行
      LD      M113  ; 工位2输送电机手动启停
      AND     M1  ; 手动方式
      ORB
      AND     X0  ; 急停信号【NC】
      AND     X6A  ; 工位1-工位2处急停
      OUT     Y8D  ; 工位二输送启停
        [note] 1-1
263   LD      L75  ; 工位2-1进托盘
      AND     M0  ; 自动运行
      LD      M116  ; 工位2-1手动进托盘
      AND     M1  ; 手动方式
      ORB
      AND     X0  ; 急停信号【NC】
      ANI     Y8F  ; 工位2-1出托盘
      ANI     X62  ; 工位2-1夹紧到位
      AND     X6A  ; 工位1-工位2处急停
      OUT     Y8E  ; 工位2-1进托盘
273   LD      L72  ; 工位2-1出货
      AND     M0  ; 自动运行
      LD      M117  ; 工位2-1手动出托盘
      AND     M1  ; 手动方式
      ORB
      AND     X0  ; 急停信号【NC】
      ANI     Y8E  ; 工位2-1进托盘
      ANI     X62  ; 工位2-1夹紧到位
      AND     X6A  ; 工位1-工位2处急停
      OUT     Y8F  ; 工位2-1出托盘
283   LD      L74  ; 工位2-1顶升进托盘上升
      OR      L77  ; 工位2-1顶升出托盘顶起
      AND     M0  ; 自动运行
      LD      M111  ; 工位2-1手动升降
      AND     M1  ; 手动方式
      ORB
      OUT     Y0C6  ; 工位2-1顶升升降
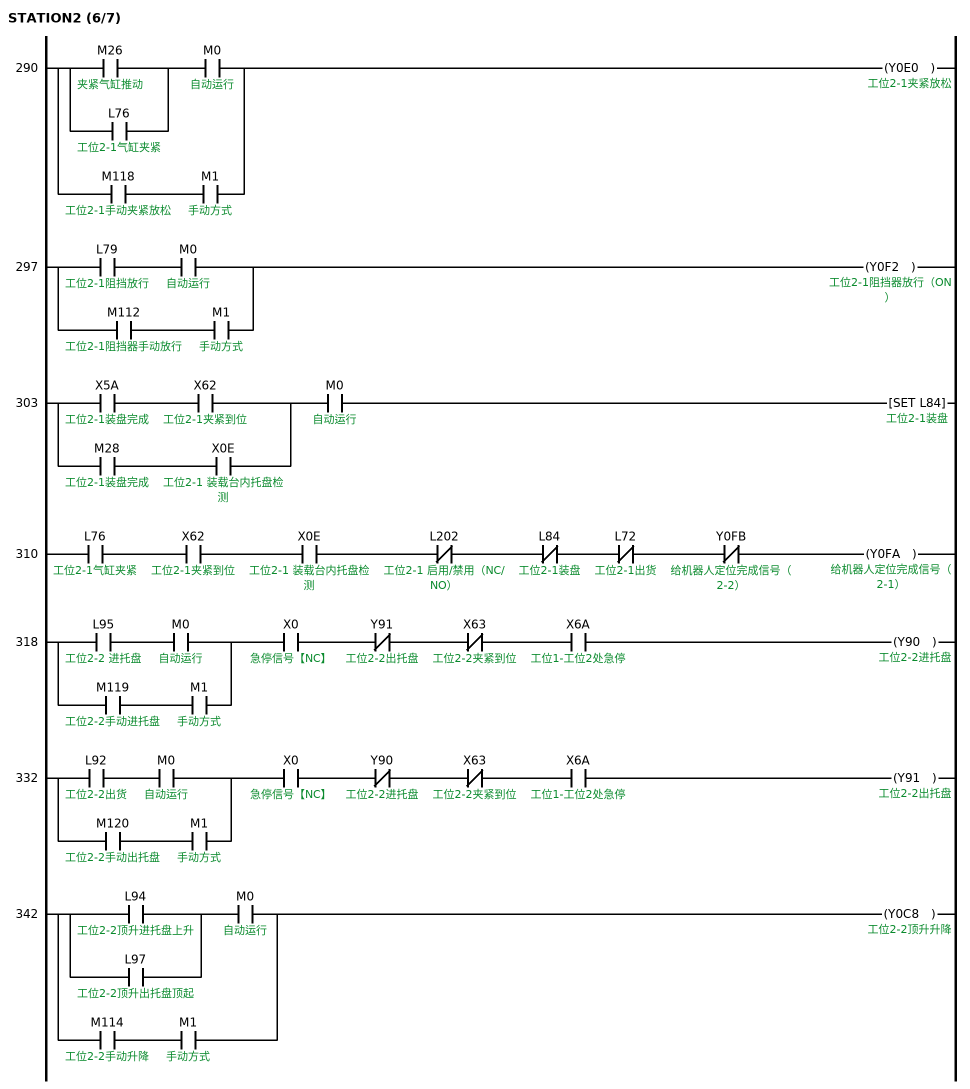
290   LD      M26  ; 夹紧气缸推动
      OR      L76  ; 工位2-1气缸夹紧
      AND     M0  ; 自动运行
      LD      M118  ; 工位2-1手动夹紧放松
      AND     M1  ; 手动方式
      ORB
      OUT     Y0E0  ; 工位2-1夹紧放松
297   LD      L79  ; 工位2-1阻挡放行
      AND     M0  ; 自动运行
      LD      M112  ; 工位2-1阻挡器手动放行
      AND     M1  ; 手动方式
      ORB
      OUT     Y0F2  ; 工位2-1阻挡器放行（ON）
303   LD      X5A  ; 工位2-1装盘完成
      AND     X62  ; 工位2-1夹紧到位
      LD      M28  ; 工位2-1装盘完成
      AND     X0E  ; 工位2-1 装载台内托盘检测
      ORB
      AND     M0  ; 自动运行
      SET     L84  ; 工位2-1装盘
310   LD      L76  ; 工位2-1气缸夹紧
      AND     X62  ; 工位2-1夹紧到位
      AND     X0E  ; 工位2-1 装载台内托盘检测
      ANI     L202  ; 工位2-1 启用/禁用（NC/NO）
      ANI     L84  ; 工位2-1装盘
      ANI     L72  ; 工位2-1出货
      ANI     Y0FB  ; 给机器人定位完成信号（2-2）
      OUT     Y0FA  ; 给机器人定位完成信号（2-1）
318   LD      L95  ; 工位2-2 进托盘
      AND     M0  ; 自动运行
      LD      M119  ; 工位2-2手动进托盘
      AND     M1  ; 手动方式
      ORB
      AND     X0  ; 急停信号【NC】
      ANI     Y91  ; 工位2-2出托盘
      ANI     X63  ; 工位2-2夹紧到位
      AND     X6A  ; 工位1-工位2处急停
      OUT     Y90  ; 工位2-2进托盘
        [note] 1-2
332   LD      L92  ; 工位2-2出货
      AND     M0  ; 自动运行
      LD      M120  ; 工位2-2手动出托盘
      AND     M1  ; 手动方式
      ORB
      AND     X0  ; 急停信号【NC】
      ANI     Y90  ; 工位2-2进托盘
      ANI     X63  ; 工位2-2夹紧到位
      AND     X6A  ; 工位1-工位2处急停
      OUT     Y91  ; 工位2-2出托盘
342   LD      L94  ; 工位2-2顶升进托盘上升
      OR      L97  ; 工位2-2顶升出托盘顶起
      AND     M0  ; 自动运行
      LD      M114  ; 工位2-2手动升降
      AND     M1  ; 手动方式
      ORB
      OUT     Y0C8  ; 工位2-2顶升升降
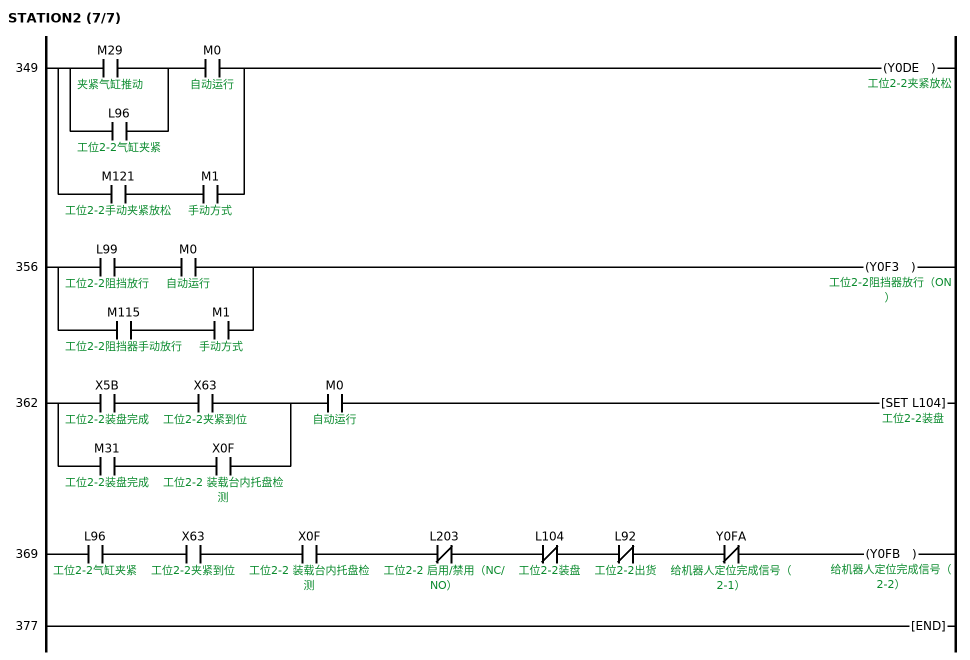
349   LD      M29  ; 夹紧气缸推动
      OR      L96  ; 工位2-2气缸夹紧
      AND     M0  ; 自动运行
      LD      M121  ; 工位2-2手动夹紧放松
      AND     M1  ; 手动方式
      ORB
      OUT     Y0DE  ; 工位2-2夹紧放松
356   LD      L99  ; 工位2-2阻挡放行
      AND     M0  ; 自动运行
      LD      M115  ; 工位2-2阻挡器手动放行
      AND     M1  ; 手动方式
      ORB
      OUT     Y0F3  ; 工位2-2阻挡器放行（ON）
362   LD      X5B  ; 工位2-2装盘完成
      AND     X63  ; 工位2-2夹紧到位
      LD      M31  ; 工位2-2装盘完成
      AND     X0F  ; 工位2-2 装载台内托盘检测
      ORB
      AND     M0  ; 自动运行
      SET     L104  ; 工位2-2装盘
369   LD      L96  ; 工位2-2气缸夹紧
      AND     X63  ; 工位2-2夹紧到位
      AND     X0F  ; 工位2-2 装载台内托盘检测
      ANI     L203  ; 工位2-2 启用/禁用（NC/NO）
      ANI     L104  ; 工位2-2装盘
      ANI     L92  ; 工位2-2出货
      ANI     Y0FA  ; 给机器人定位完成信号（2-1）
      OUT     Y0FB  ; 给机器人定位完成信号（2-2）
377   END
END_PROGRAM

PROGRAM STATION3
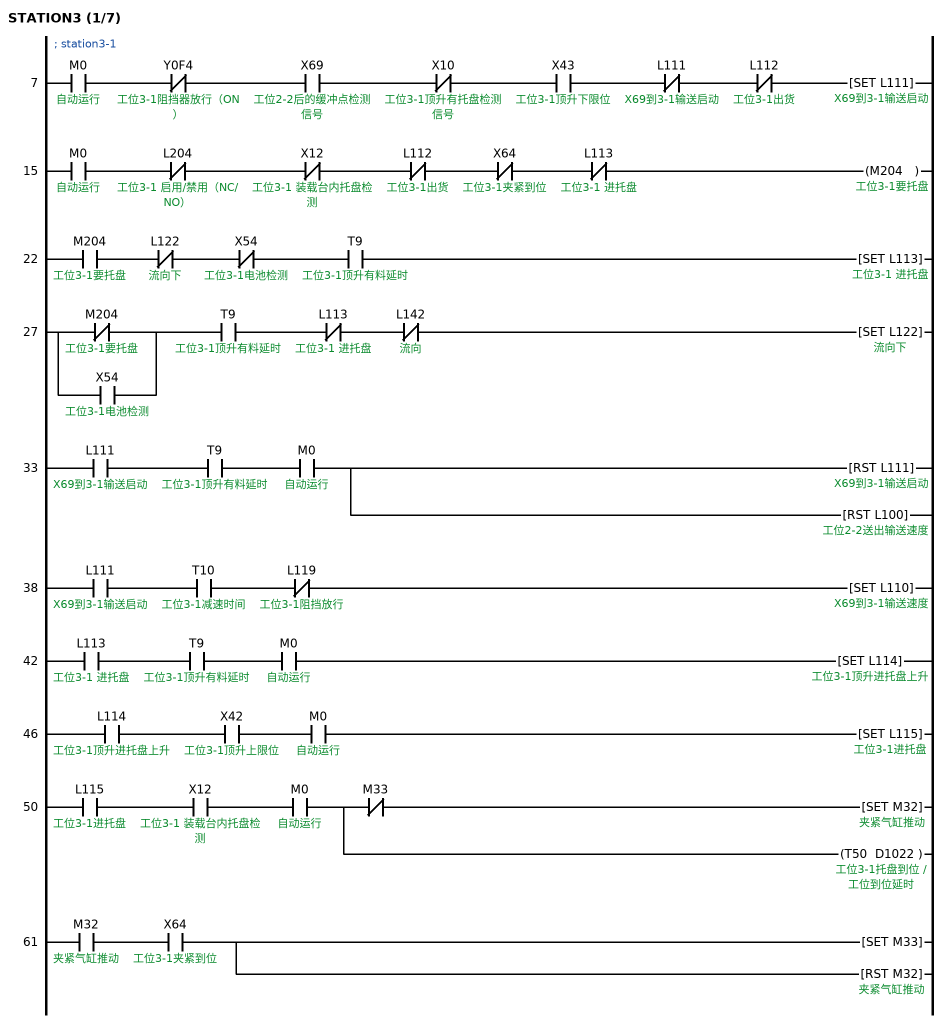
; station3-1
7     LD      M0  ; 自动运行
      ANI     Y0F4  ; 工位3-1阻挡器放行（ON）
      AND     X69  ; 工位2-2后的缓冲点检测信号
      ANI     X10  ; 工位3-1顶升有托盘检测信号
      AND     X43  ; 工位3-1顶升下限位
      ANI     L111  ; X69到3-1输送启动
      ANI     L112  ; 工位3-1出货
      SET     L111  ; X69到3-1输送启动
15    LD      M0  ; 自动运行
      ANI     L204  ; 工位3-1 启用/禁用（NC/NO）
      ANI     X12  ; 工位3-1 装载台内托盘检测
      ANI     L112  ; 工位3-1出货
      ANI     X64  ; 工位3-1夹紧到位
      ANI     L113  ; 工位3-1 进托盘
      OUT     M204  ; 工位3-1要托盘
22    LD      M204  ; 工位3-1要托盘
      ANI     L122  ; 流向下
      ANI     X54  ; 工位3-1电池检测
      AND     T9  ; 工位3-1顶升有料延时
      SET     L113  ; 工位3-1 进托盘
27    LDI     M204  ; 工位3-1要托盘
      OR      X54  ; 工位3-1电池检测
      AND     T9  ; 工位3-1顶升有料延时
      ANI     L113  ; 工位3-1 进托盘
      ANI     L142  ; 流向
      SET     L122  ; 流向下
33    LD      L111  ; X69到3-1输送启动
      AND     T9  ; 工位3-1顶升有料延时
      AND     M0  ; 自动运行
      RST     L111  ; X69到3-1输送启动
      RST     L100  ; 工位2-2送出输送速度
38    LD      L111  ; X69到3-1输送启动
      AND     T10  ; 工位3-1减速时间
      ANI     L119  ; 工位3-1阻挡放行
      SET     L110  ; X69到3-1输送速度
42    LD      L113  ; 工位3-1 进托盘
      AND     T9  ; 工位3-1顶升有料延时
      AND     M0  ; 自动运行
      SET     L114  ; 工位3-1顶升进托盘上升
46    LD      L114  ; 工位3-1顶升进托盘上升
      AND     X42  ; 工位3-1顶升上限位
      AND     M0  ; 自动运行
      SET     L115  ; 工位3-1进托盘
50    LD      L115  ; 工位3-1进托盘
      AND     X12  ; 工位3-1 装载台内托盘检测
      AND     M0  ; 自动运行
      MPS
      ANI     M33
      SET     M32  ; 夹紧气缸推动
      MPP
      OUT     T50 D1022  ; 工位3-1托盘到位 / 工位到位延时
61    LD      M32  ; 夹紧气缸推动
      AND     X64  ; 工位3-1夹紧到位
      SET     M33
      RST     M32  ; 夹紧气缸推动
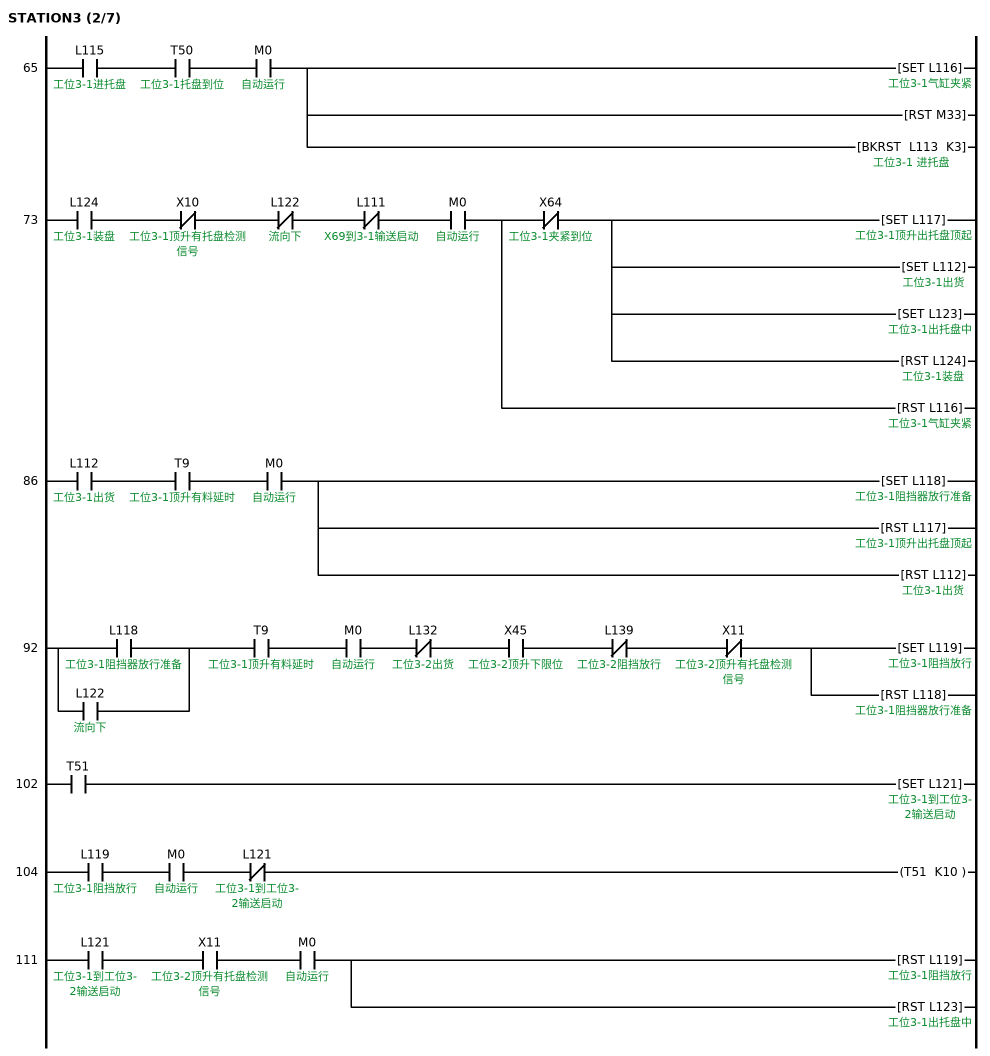
65    LD      L115  ; 工位3-1进托盘
      AND     T50  ; 工位3-1托盘到位
      AND     M0  ; 自动运行
      SET     L116  ; 工位3-1气缸夹紧
      RST     M33
      BKRST   L113 K3
73    LD      L124  ; 工位3-1装盘
      ANI     X10  ; 工位3-1顶升有托盘检测信号
      ANI     L122  ; 流向下
      ANI     L111  ; X69到3-1输送启动
      AND     M0  ; 自动运行
      MPS
      ANI     X64  ; 工位3-1夹紧到位
      SET     L117  ; 工位3-1顶升出托盘顶起
      SET     L112  ; 工位3-1出货
      SET     L123  ; 工位3-1出托盘中
      RST     L124  ; 工位3-1装盘
      MPP
      RST     L116  ; 工位3-1气缸夹紧
86    LD      L112  ; 工位3-1出货
      AND     T9  ; 工位3-1顶升有料延时
      AND     M0  ; 自动运行
      SET     L118  ; 工位3-1阻挡器放行准备
      RST     L117  ; 工位3-1顶升出托盘顶起
      RST     L112  ; 工位3-1出货
92    LD      L118  ; 工位3-1阻挡器放行准备
      OR      L122  ; 流向下
      AND     T9  ; 工位3-1顶升有料延时
      AND     M0  ; 自动运行
      ANI     L132  ; 工位3-2出货
      AND     X45  ; 工位3-2顶升下限位
      ANI     L139  ; 工位3-2阻挡放行
      ANI     X11  ; 工位3-2顶升有托盘检测信号
      SET     L119  ; 工位3-1阻挡放行
      RST     L118  ; 工位3-1阻挡器放行准备
102   LD      T51
      SET     L121  ; 工位3-1到工位3-2输送启动
104   LD      L119  ; 工位3-1阻挡放行
      AND     M0  ; 自动运行
      ANI     L121  ; 工位3-1到工位3-2输送启动
      OUT     T51 K10
111   LD      L121  ; 工位3-1到工位3-2输送启动
      AND     X11  ; 工位3-2顶升有托盘检测信号
      AND     M0  ; 自动运行
      RST     L119  ; 工位3-1阻挡放行
      RST     L123  ; 工位3-1出托盘中
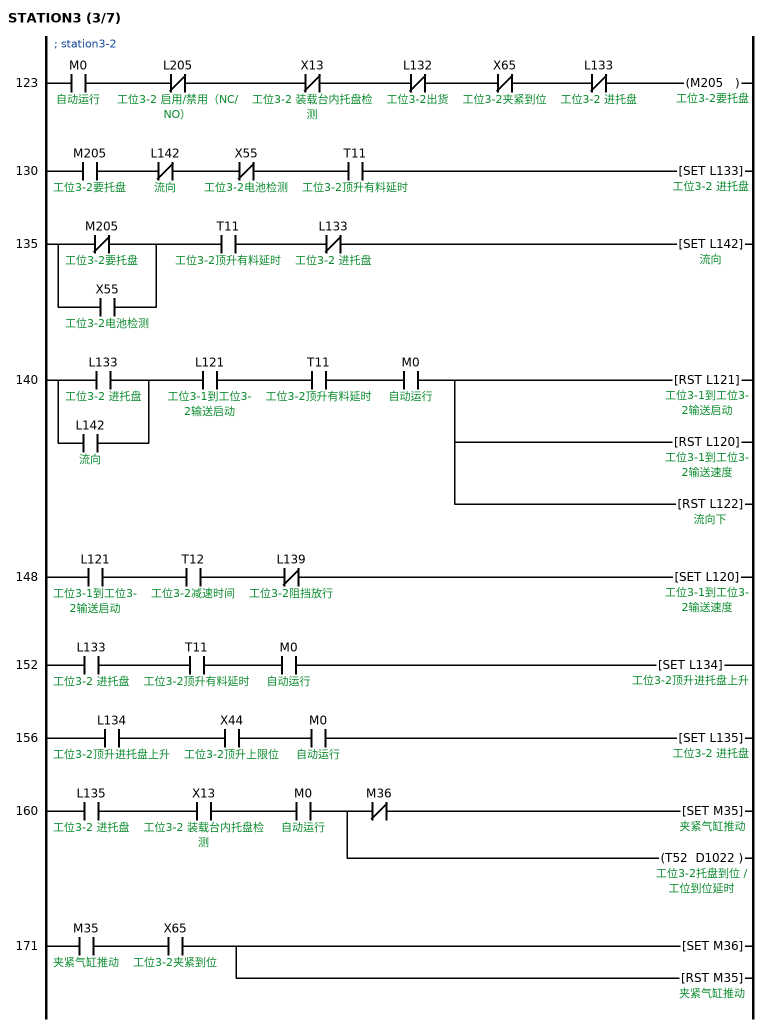
; station3-2
123   LD      M0  ; 自动运行
      ANI     L205  ; 工位3-2 启用/禁用（NC/NO）
      ANI     X13  ; 工位3-2 装载台内托盘检测
      ANI     L132  ; 工位3-2出货
      ANI     X65  ; 工位3-2夹紧到位
      ANI     L133  ; 工位3-2 进托盘
      OUT     M205  ; 工位3-2要托盘
130   LD      M205  ; 工位3-2要托盘
      ANI     L142  ; 流向
      ANI     X55  ; 工位3-2电池检测
      AND     T11  ; 工位3-2顶升有料延时
      SET     L133  ; 工位3-2 进托盘
135   LDI     M205  ; 工位3-2要托盘
      OR      X55  ; 工位3-2电池检测
      AND     T11  ; 工位3-2顶升有料延时
      ANI     L133  ; 工位3-2 进托盘
      SET     L142  ; 流向
140   LD      L133  ; 工位3-2 进托盘
      OR      L142  ; 流向
      AND     L121  ; 工位3-1到工位3-2输送启动
      AND     T11  ; 工位3-2顶升有料延时
      AND     M0  ; 自动运行
      RST     L121  ; 工位3-1到工位3-2输送启动
      RST     L120  ; 工位3-1到工位3-2输送速度
      RST     L122  ; 流向下
148   LD      L121  ; 工位3-1到工位3-2输送启动
      AND     T12  ; 工位3-2减速时间
      ANI     L139  ; 工位3-2阻挡放行
      SET     L120  ; 工位3-1到工位3-2输送速度
152   LD      L133  ; 工位3-2 进托盘
      AND     T11  ; 工位3-2顶升有料延时
      AND     M0  ; 自动运行
      SET     L134  ; 工位3-2顶升进托盘上升
156   LD      L134  ; 工位3-2顶升进托盘上升
      AND     X44  ; 工位3-2顶升上限位
      AND     M0  ; 自动运行
      SET     L135  ; 工位3-2 进托盘
160   LD      L135  ; 工位3-2 进托盘
      AND     X13  ; 工位3-2 装载台内托盘检测
      AND     M0  ; 自动运行
      MPS
      ANI     M36
      SET     M35  ; 夹紧气缸推动
      MPP
      OUT     T52 D1022  ; 工位3-2托盘到位 / 工位到位延时
171   LD      M35  ; 夹紧气缸推动
      AND     X65  ; 工位3-2夹紧到位
      SET     M36
      RST     M35  ; 夹紧气缸推动
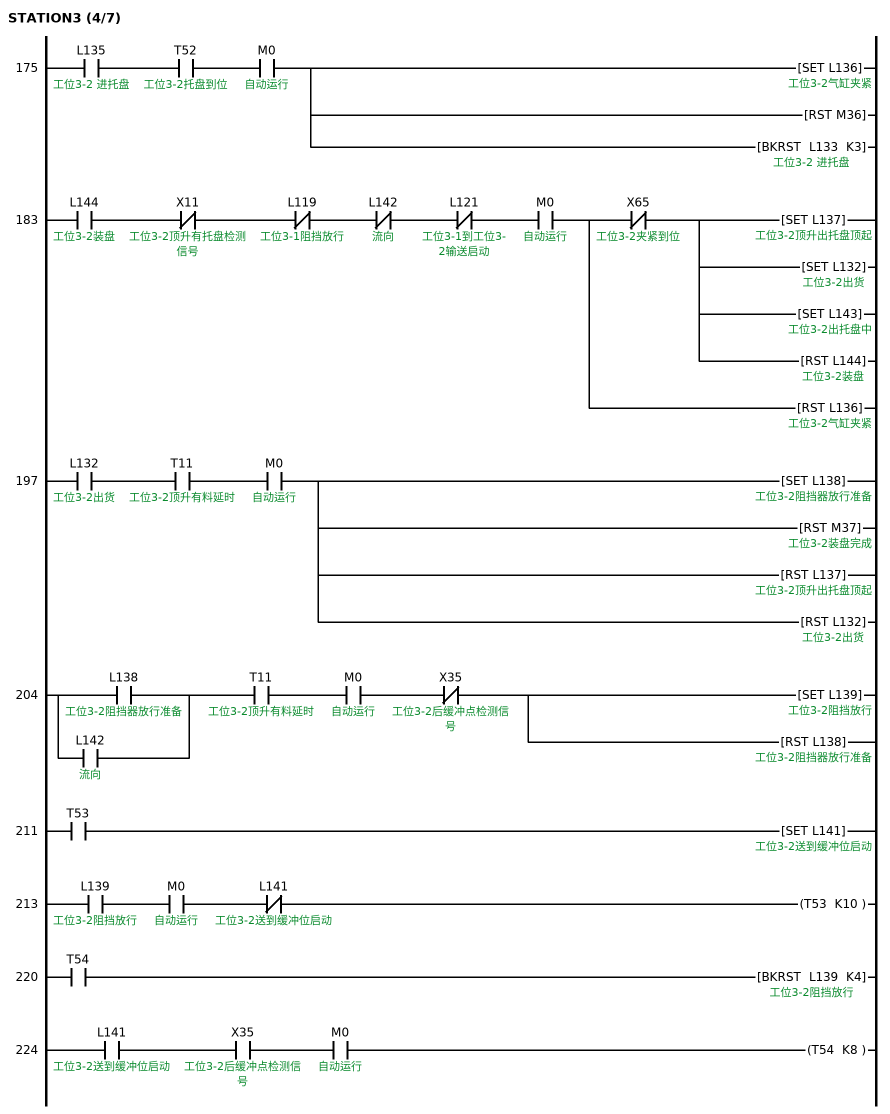
175   LD      L135  ; 工位3-2 进托盘
      AND     T52  ; 工位3-2托盘到位
      AND     M0  ; 自动运行
      SET     L136  ; 工位3-2气缸夹紧
      RST     M36
      BKRST   L133 K3
183   LD      L144  ; 工位3-2装盘
      ANI     X11  ; 工位3-2顶升有托盘检测信号
      ANI     L119  ; 工位3-1阻挡放行
      ANI     L142  ; 流向
      ANI     L121  ; 工位3-1到工位3-2输送启动
      AND     M0  ; 自动运行
      MPS
      ANI     X65  ; 工位3-2夹紧到位
      SET     L137  ; 工位3-2顶升出托盘顶起
      SET     L132  ; 工位3-2出货
      SET     L143  ; 工位3-2出托盘中
      RST     L144  ; 工位3-2装盘
      MPP
      RST     L136  ; 工位3-2气缸夹紧
197   LD      L132  ; 工位3-2出货
      AND     T11  ; 工位3-2顶升有料延时
      AND     M0  ; 自动运行
      SET     L138  ; 工位3-2阻挡器放行准备
      RST     M37  ; 工位3-2装盘完成
      RST     L137  ; 工位3-2顶升出托盘顶起
      RST     L132  ; 工位3-2出货
204   LD      L138  ; 工位3-2阻挡器放行准备
      OR      L142  ; 流向
      AND     T11  ; 工位3-2顶升有料延时
      AND     M0  ; 自动运行
      ANI     X35  ; 工位3-2后缓冲点检测信号
      SET     L139  ; 工位3-2阻挡放行
      RST     L138  ; 工位3-2阻挡器放行准备
211   LD      T53
      SET     L141  ; 工位3-2送到缓冲位启动
213   LD      L139  ; 工位3-2阻挡放行
      AND     M0  ; 自动运行
      ANI     L141  ; 工位3-2送到缓冲位启动
      OUT     T53 K10
220   LD      T54
      BKRST   L139 K4
224   LD      L141  ; 工位3-2送到缓冲位启动
      AND     X35  ; 工位3-2后缓冲点检测信号
      AND     M0  ; 自动运行
      OUT     T54 K8
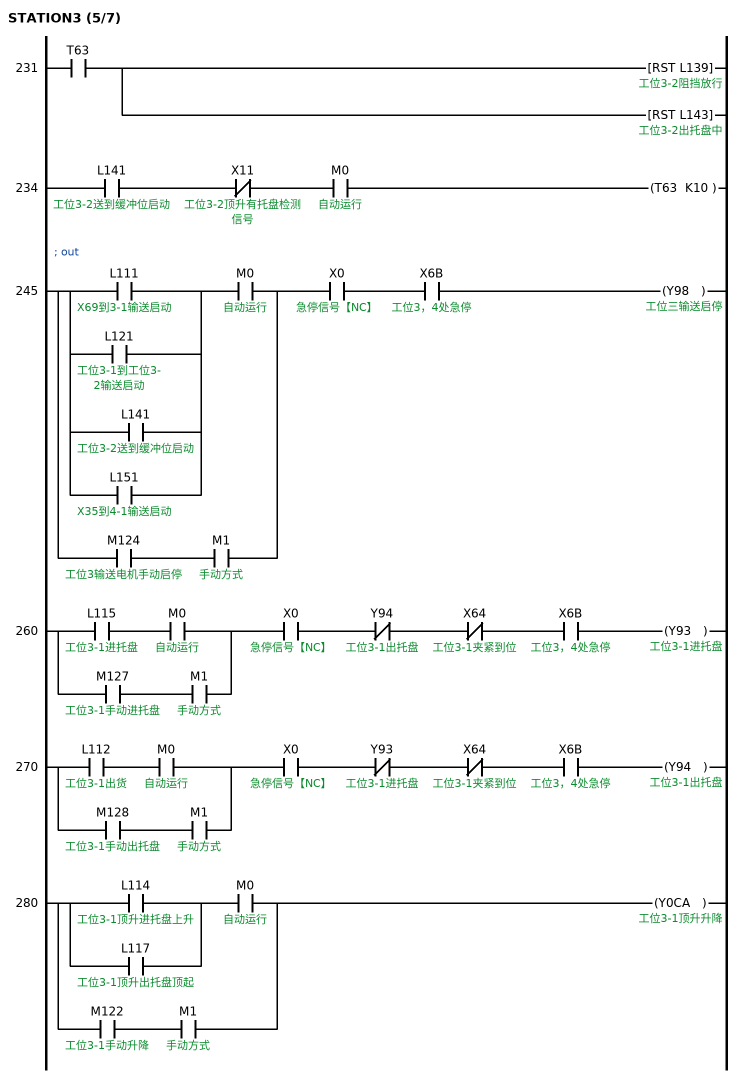
231   LD      T63
      RST     L139  ; 工位3-2阻挡放行
      RST     L143  ; 工位3-2出托盘中
234   LD      L141  ; 工位3-2送到缓冲位启动
      ANI     X11  ; 工位3-2顶升有托盘检测信号
      AND     M0  ; 自动运行
      OUT     T63 K10
; out
245   LD      L111  ; X69到3-1输送启动
      OR      L121  ; 工位3-1到工位3-2输送启动
      OR      L141  ; 工位3-2送到缓冲位启动
      OR      L151  ; X35到4-1输送启动
      AND     M0  ; 自动运行
      LD      M124  ; 工位3输送电机手动启停
      AND     M1  ; 手动方式
      ORB
      AND     X0  ; 急停信号【NC】
      AND     X6B  ; 工位3，4处急停
      OUT     Y98  ; 工位三输送启停
        [note] 3-1
260   LD      L115  ; 工位3-1进托盘
      AND     M0  ; 自动运行
      LD      M127  ; 工位3-1手动进托盘
      AND     M1  ; 手动方式
      ORB
      AND     X0  ; 急停信号【NC】
      ANI     Y94  ; 工位3-1出托盘
      ANI     X64  ; 工位3-1夹紧到位
      AND     X6B  ; 工位3，4处急停
      OUT     Y93  ; 工位3-1进托盘
270   LD      L112  ; 工位3-1出货
      AND     M0  ; 自动运行
      LD      M128  ; 工位3-1手动出托盘
      AND     M1  ; 手动方式
      ORB
      AND     X0  ; 急停信号【NC】
      ANI     Y93  ; 工位3-1进托盘
      ANI     X64  ; 工位3-1夹紧到位
      AND     X6B  ; 工位3，4处急停
      OUT     Y94  ; 工位3-1出托盘
280   LD      L114  ; 工位3-1顶升进托盘上升
      OR      L117  ; 工位3-1顶升出托盘顶起
      AND     M0  ; 自动运行
      LD      M122  ; 工位3-1手动升降
      AND     M1  ; 手动方式
      ORB
      OUT     Y0CA  ; 工位3-1顶升升降
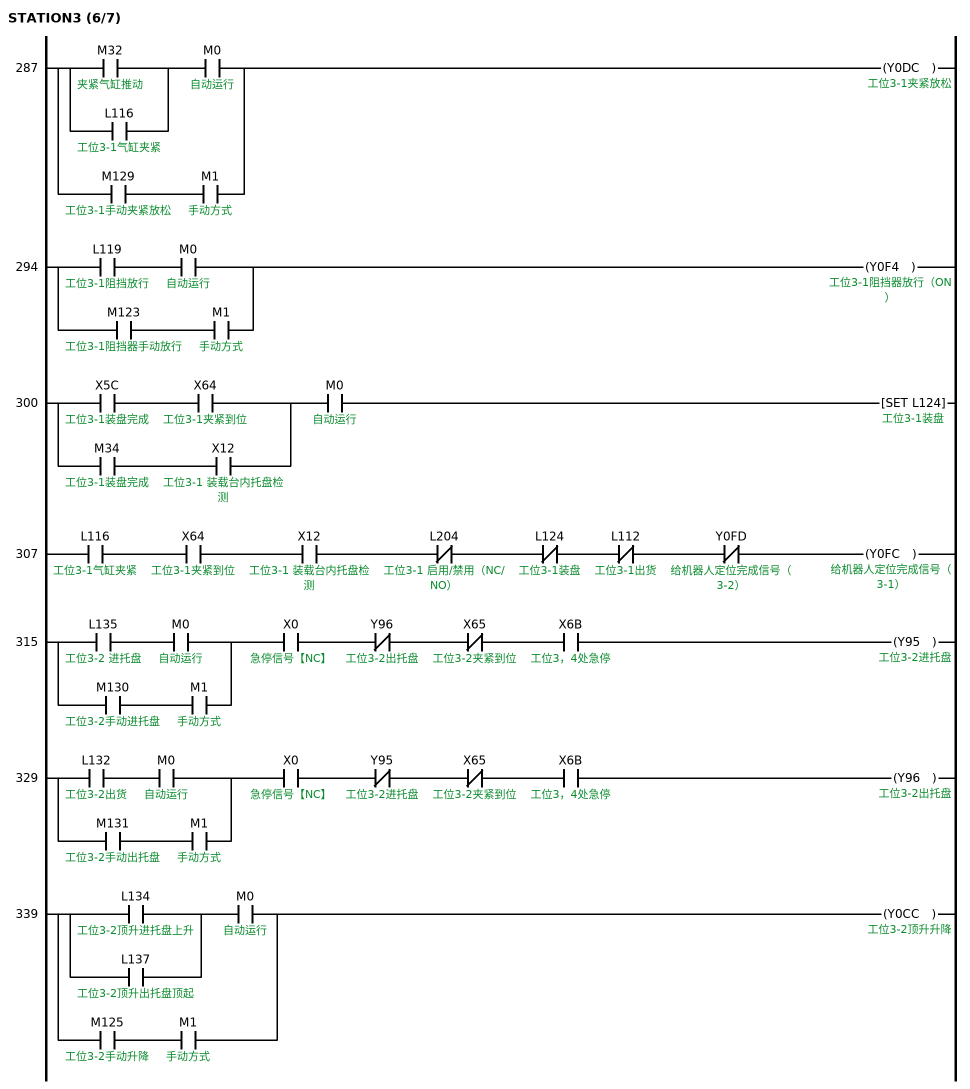
287   LD      M32  ; 夹紧气缸推动
      OR      L116  ; 工位3-1气缸夹紧
      AND     M0  ; 自动运行
      LD      M129  ; 工位3-1手动夹紧放松
      AND     M1  ; 手动方式
      ORB
      OUT     Y0DC  ; 工位3-1夹紧放松
294   LD      L119  ; 工位3-1阻挡放行
      AND     M0  ; 自动运行
      LD      M123  ; 工位3-1阻挡器手动放行
      AND     M1  ; 手动方式
      ORB
      OUT     Y0F4  ; 工位3-1阻挡器放行（ON）
300   LD      X5C  ; 工位3-1装盘完成
      AND     X64  ; 工位3-1夹紧到位
      LD      M34  ; 工位3-1装盘完成
      AND     X12  ; 工位3-1 装载台内托盘检测
      ORB
      AND     M0  ; 自动运行
      SET     L124  ; 工位3-1装盘
307   LD      L116  ; 工位3-1气缸夹紧
      AND     X64  ; 工位3-1夹紧到位
      AND     X12  ; 工位3-1 装载台内托盘检测
      ANI     L204  ; 工位3-1 启用/禁用（NC/NO）
      ANI     L124  ; 工位3-1装盘
      ANI     L112  ; 工位3-1出货
      ANI     Y0FD  ; 给机器人定位完成信号（3-2）
      OUT     Y0FC  ; 给机器人定位完成信号（3-1）
315   LD      L135  ; 工位3-2 进托盘
      AND     M0  ; 自动运行
      LD      M130  ; 工位3-2手动进托盘
      AND     M1  ; 手动方式
      ORB
      AND     X0  ; 急停信号【NC】
      ANI     Y96  ; 工位3-2出托盘
      ANI     X65  ; 工位3-2夹紧到位
      AND     X6B  ; 工位3，4处急停
      OUT     Y95  ; 工位3-2进托盘
        [note] 3-2
329   LD      L132  ; 工位3-2出货
      AND     M0  ; 自动运行
      LD      M131  ; 工位3-2手动出托盘
      AND     M1  ; 手动方式
      ORB
      AND     X0  ; 急停信号【NC】
      ANI     Y95  ; 工位3-2进托盘
      ANI     X65  ; 工位3-2夹紧到位
      AND     X6B  ; 工位3，4处急停
      OUT     Y96  ; 工位3-2出托盘
339   LD      L134  ; 工位3-2顶升进托盘上升
      OR      L137  ; 工位3-2顶升出托盘顶起
      AND     M0  ; 自动运行
      LD      M125  ; 工位3-2手动升降
      AND     M1  ; 手动方式
      ORB
      OUT     Y0CC  ; 工位3-2顶升升降
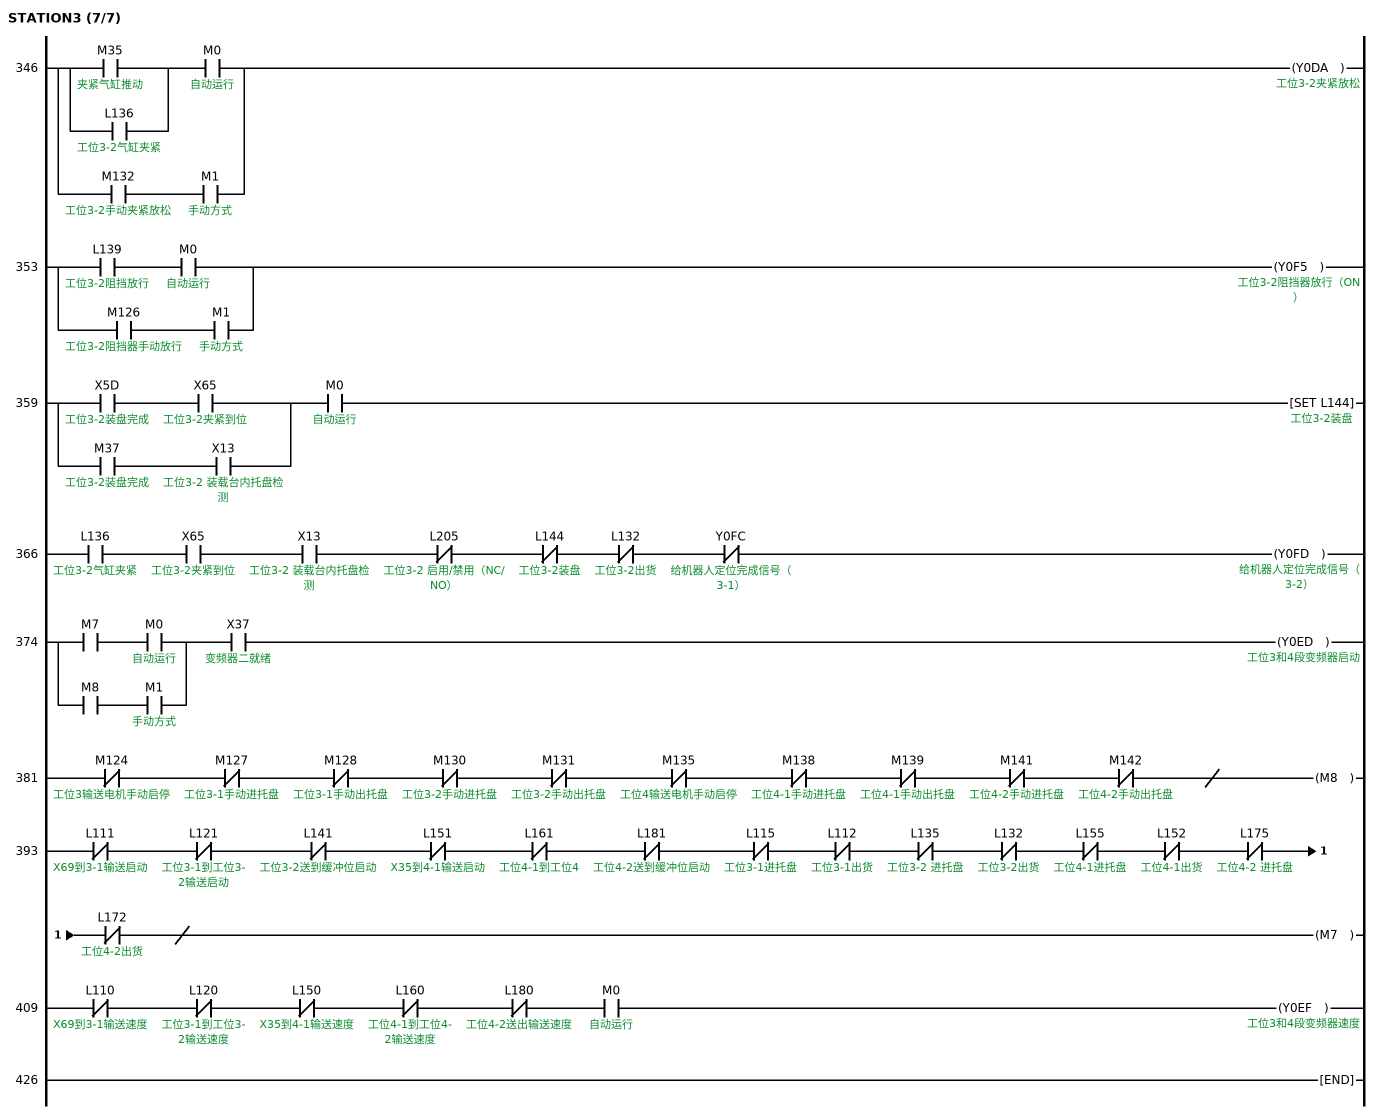
346   LD      M35  ; 夹紧气缸推动
      OR      L136  ; 工位3-2气缸夹紧
      AND     M0  ; 自动运行
      LD      M132  ; 工位3-2手动夹紧放松
      AND     M1  ; 手动方式
      ORB
      OUT     Y0DA  ; 工位3-2夹紧放松
353   LD      L139  ; 工位3-2阻挡放行
      AND     M0  ; 自动运行
      LD      M126  ; 工位3-2阻挡器手动放行
      AND     M1  ; 手动方式
      ORB
      OUT     Y0F5  ; 工位3-2阻挡器放行（ON）
359   LD      X5D  ; 工位3-2装盘完成
      AND     X65  ; 工位3-2夹紧到位
      LD      M37  ; 工位3-2装盘完成
      AND     X13  ; 工位3-2 装载台内托盘检测
      ORB
      AND     M0  ; 自动运行
      SET     L144  ; 工位3-2装盘
366   LD      L136  ; 工位3-2气缸夹紧
      AND     X65  ; 工位3-2夹紧到位
      AND     X13  ; 工位3-2 装载台内托盘检测
      ANI     L205  ; 工位3-2 启用/禁用（NC/NO）
      ANI     L144  ; 工位3-2装盘
      ANI     L132  ; 工位3-2出货
      ANI     Y0FC  ; 给机器人定位完成信号（3-1）
      OUT     Y0FD  ; 给机器人定位完成信号（3-2）
374   LD      M7
      AND     M0  ; 自动运行
      LD      M8
      AND     M1  ; 手动方式
      ORB
      AND     X37  ; 变频器二就绪
      OUT     Y0ED  ; 工位3和4段变频器启动
381   LDI     M124  ; 工位3输送电机手动启停
      ANI     M127  ; 工位3-1手动进托盘
      ANI     M128  ; 工位3-1手动出托盘
      ANI     M130  ; 工位3-2手动进托盘
      ANI     M131  ; 工位3-2手动出托盘
      ANI     M135  ; 工位4输送电机手动启停
      ANI     M138  ; 工位4-1手动进托盘
      ANI     M139  ; 工位4-1手动出托盘
      ANI     M141  ; 工位4-2手动进托盘
      ANI     M142  ; 工位4-2手动出托盘
      INV
      OUT     M8
393   LDI     L111  ; X69到3-1输送启动
      ANI     L121  ; 工位3-1到工位3-2输送启动
      ANI     L141  ; 工位3-2送到缓冲位启动
      ANI     L151  ; X35到4-1输送启动
      ANI     L161  ; 工位4-1到工位4
      ANI     L181  ; 工位4-2送到缓冲位启动
      ANI     L115  ; 工位3-1进托盘
      ANI     L112  ; 工位3-1出货
      ANI     L135  ; 工位3-2 进托盘
      ANI     L132  ; 工位3-2出货
      ANI     L155  ; 工位4-1进托盘
      ANI     L152  ; 工位4-1出货
      ANI     L175  ; 工位4-2 进托盘
      ANI     L172  ; 工位4-2出货
      INV
      OUT     M7
409   LDI     L110  ; X69到3-1输送速度
      ANI     L120  ; 工位3-1到工位3-2输送速度
      ANI     L150  ; X35到4-1输送速度
      ANI     L160  ; 工位4-1到工位4-2输送速度
      ANI     L180  ; 工位4-2送出输送速度
      AND     M0  ; 自动运行
      OUT     Y0EF  ; 工位3和4段变频器速度
        [note] ON高速，OFF低速
426   END
END_PROGRAM

PROGRAM STATION4
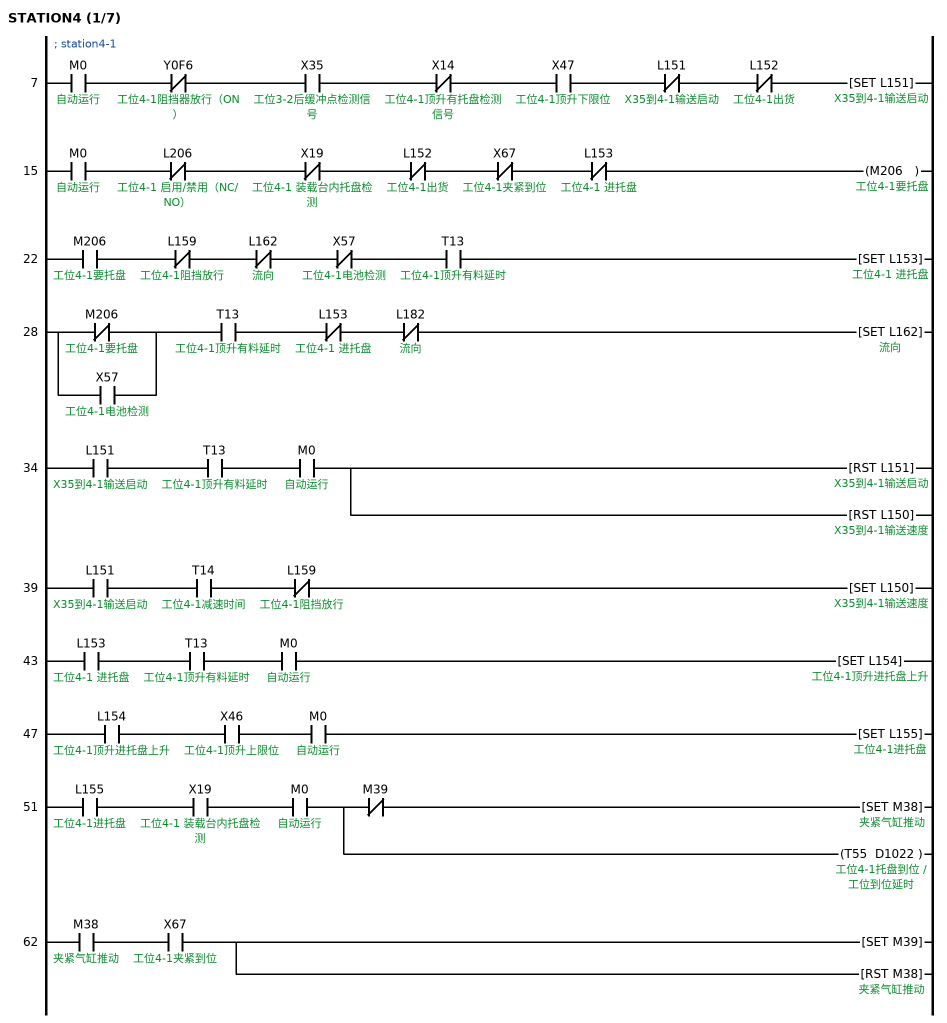
; station4-1
7     LD      M0  ; 自动运行
      ANI     Y0F6  ; 工位4-1阻挡器放行（ON）
      AND     X35  ; 工位3-2后缓冲点检测信号
      ANI     X14  ; 工位4-1顶升有托盘检测信号
      AND     X47  ; 工位4-1顶升下限位
      ANI     L151  ; X35到4-1输送启动
      ANI     L152  ; 工位4-1出货
      SET     L151  ; X35到4-1输送启动
15    LD      M0  ; 自动运行
      ANI     L206  ; 工位4-1 启用/禁用（NC/NO）
      ANI     X19  ; 工位4-1 装载台内托盘检测
      ANI     L152  ; 工位4-1出货
      ANI     X67  ; 工位4-1夹紧到位
      ANI     L153  ; 工位4-1 进托盘
      OUT     M206  ; 工位4-1要托盘
22    LD      M206  ; 工位4-1要托盘
      ANI     L159  ; 工位4-1阻挡放行
      ANI     L162  ; 流向
      ANI     X57  ; 工位4-1电池检测
      AND     T13  ; 工位4-1顶升有料延时
      SET     L153  ; 工位4-1 进托盘
28    LDI     M206  ; 工位4-1要托盘
      OR      X57  ; 工位4-1电池检测
      AND     T13  ; 工位4-1顶升有料延时
      ANI     L153  ; 工位4-1 进托盘
      ANI     L182  ; 流向
      SET     L162  ; 流向
34    LD      L151  ; X35到4-1输送启动
      AND     T13  ; 工位4-1顶升有料延时
      AND     M0  ; 自动运行
      RST     L151  ; X35到4-1输送启动
      RST     L150  ; X35到4-1输送速度
39    LD      L151  ; X35到4-1输送启动
      AND     T14  ; 工位4-1减速时间
      ANI     L159  ; 工位4-1阻挡放行
      SET     L150  ; X35到4-1输送速度
43    LD      L153  ; 工位4-1 进托盘
      AND     T13  ; 工位4-1顶升有料延时
      AND     M0  ; 自动运行
      SET     L154  ; 工位4-1顶升进托盘上升
47    LD      L154  ; 工位4-1顶升进托盘上升
      AND     X46  ; 工位4-1顶升上限位
      AND     M0  ; 自动运行
      SET     L155  ; 工位4-1进托盘
51    LD      L155  ; 工位4-1进托盘
      AND     X19  ; 工位4-1 装载台内托盘检测
      AND     M0  ; 自动运行
      MPS
      ANI     M39
      SET     M38  ; 夹紧气缸推动
      MPP
      OUT     T55 D1022  ; 工位4-1托盘到位 / 工位到位延时
62    LD      M38  ; 夹紧气缸推动
      AND     X67  ; 工位4-1夹紧到位
      SET     M39
      RST     M38  ; 夹紧气缸推动
